(* IEC 61131-3 sources: elnaProjects/kc6/build_BaseProject_ecl/_ (part 2) *)

  StrAlg.CanRun := StrAlg.inCanRun;
  StrAlg.OpcCommandsDisabled := StrAlg.inOpcCommandsDisabled;

  IF StrAlg.isRuning THEN

      StrAlg.hasError := pnsOff.error OR nu1Off.error OR nu2Off.error
      OR stopNU1.error OR stopNU2.error OR testUnsuccessful.error;

      IF puskOilSystem.top THEN
           askQuestion(algContinue);
      END_IF;

      IF algContinue.answer = _Answers.ANS_YES AND NOT nuOff.top THEN

          runPhase(nuOff);

          IF Im.nu1.onStatus = _statusDualInput.STATUS_ON THEN
  		runPhase(nu1Off);
          END_IF;

          IF Im.nu2.onStatus = _statusDualInput.STATUS_ON THEN
  		runPhase(nu2Off);
          END_IF;

      END_IF;

      IF nuOff.start AND NOT nuOff.top THEN
            runPhase(BreakTest);
  	nuOff.top:= Im.nu1.onStatus = _statusDualInput.STATUS_Off
                    AND Im.nu2.onStatus = _statusDualInput.STATUS_Off;
      END_IF;

      IF nuOff.top THEN

          runPhase(dPmgAi);
          runPhase(dPmgDi);
      END_IF;

      IF dPmgDi.start AND NOT dPmgDi.top THEN
          dPmgDi.top:=Im.SingleSignals.dP_maslo_gaz_menshe_100_kPa.q;
      END_IF;

      IF dPmgAi.top AND dPmgDi.top THEN
          runPhase(nuOn);
          runPhase(noRezrv);
      END_IF;

      IF noRezrv.start AND NOT noRezrv.top THEN
          noRezrv.top:=NotHasRezervNU;
      END_IF;

       IF nuOn.start AND (NOT WaitOnNU.Q) THEN
          WaitOnNU(IN:=Im.nu1.onStatus = _statusDualInput.STATUS_On OR
              Im.nu2.onStatus = _statusDualInput.STATUS_On, PT:=T#1S);
          nuOn.top:=Im.nu1.onStatus = _statusDualInput.STATUS_On OR
              Im.nu2.onStatus = _statusDualInput.STATUS_On;
      END_IF;

      IF  WaitOnNU.Q AND noRezrv.top THEN
          ai.Perepad_davleniya_maslo_gaz.Disabled_LA:=TRUE;
          ai.Perepad_davleniya_maslo_gaz.Disabled_LW:=TRUE;
          ai.Davlenie_masla_smazki_nizkoe.Disabled_LA:=TRUE;
          ai.Davlenie_masla_smazki_nizkoe.Disabled_LW:=TRUE;
          ai.Davlenie_masla_smazki_visokoe.Disabled_LW:=TRUE;

          resetAiProtection(protections.Davlenie_masla_smazki_nizkoe_LA);
          resetAiProtection(protections.Perepad_davleniya_maslo_gaz_LA);
          resetDiProtection(protections.dP_maslo_gaz_menshe_100_kPa_DI);

          resetIfRunning(algoritms.autoNu);
          resetIfRunning(algoritms.AutoPns);

          runPhase(stopANU);
          runPhase(pnsOff);

          runPhase(stopNU1);
          runPhase(stopNU2);

      END_IF;

      IF stopANU.start AND NOT stopANU.top THEN

  	stopANU.top:= Im.nu1.onStatus = _statusDualInput.STATUS_Off AND
                          Im.nu2.onStatus = _statusDualInput.STATUS_Off;
      END_IF;

      IF BreakTest.top AND NOT pnsOff.top THEN
  	testUnsuccessful.error:=TRUE;
      END_IF;

      IF pnsOff.top AND stopANU.top THEN
            resetPhase(BreakTest);
  	waitReset(IN:=TRUE, PT:= T#3S);
      END_IF;

      IF waitReset.Q THEN
          algManager.nMode:=ModeGpa.MODE_STOP;
          resetIfRunning(StrAlg);
      END_IF;

      StrAlg.isEnded:= pnsOff.top AND stopANU.top;

  END_IF;

  StrAlg.CanRun := StrAlg.inCanRun;
  StrAlg.OpcCommandsDisabled := StrAlg.inOpcCommandsDisabled;

  (* ---- Если управление с ВУ заблокировано, то  передаем команду из алгоритма ---- *)
  IF StrAlg.inOpcCommandsDisabled THEN
  	StrAlg.inCommand := StrAlg.inCommand_Alg;
  ELSE (* иначе передаем команду с АРМа*)
  	StrAlg.inCommand := StrAlg.inCommand_ARM;
  END_IF;

  _sunpackerCommand(command := StrAlg.inCommand);
  	source := _sunpackerCommand.source;
  	cmd := _sunpackerCommand.cmd;

  IF cmd <> 0 AND lastCmd <> cmd AND (((NOT StrAlg.opcCommandsDisabled) AND source > 0) OR source = 0) then
  	CASE BYTE_TO_INT(cmd) OF
  		(*cmdRun*) 1: 	IF (StrAlg.CanRun) THEN
  					StrAlg.isRuning := TRUE;
  					StrAlg.isEnded := FALSE;
  					StrAlg.hasError := FALSE;
  					(*****************       OnRun       *****************)

                                                    algManager.nMode:=ModeGpa.MODE_TESTDPMG;
                                                    algoritms.puskOilSystem.inCanRun:= TRUE;
                                                    runPhase(puskOilSystem);

  					cmd_for_Status := cmd;
  					source_for_Status := source;
  					command_error_for_Status := 0;
  				ELSE
  					StrAlg.isRuning := FALSE;
  					StrAlg.isEnded := FALSE;
  					StrAlg.hasError 	:= FALSE;

  					cmd_for_Status := 0;
  					source_for_Status := source;
  					command_error_for_Status := cmd;
  				END_IF;
  		(*cmdReset*) 2: 	StrAlg.isRuning := FALSE;
  				StrAlg.isEnded := FALSE;
  				StrAlg.hasError 	:= FALSE;

                                           (*****************       OnReset       *****************)
                                          waitReset(IN:=FALSE);
                                          WaitOnNU(IN:=FALSE);

                                          ai.Davlenie_masla_smazki_nizkoe.Disabled_LA:=TRUE;
                                          ai.Davlenie_masla_smazki_nizkoe.Disabled_LW:=TRUE;
                                          ai.Davlenie_masla_smazki_visokoe.Disabled_LW:=TRUE;
                                          resetAiProtection(protections.Davlenie_masla_smazki_nizkoe_LA);
                                          resetAiProtection(protections.Perepad_davleniya_maslo_gaz_LA);
                                          resetDiProtection(protections.dP_maslo_gaz_menshe_100_kPa_DI);

                                          resetPhase(puskOilSystem);
                                          resetPhase(nuOff);
                                          resetPhase(dPmgAi);
                                          resetPhase(dPmgDi);
                                          resetPhase(nuOn);
                                          resetPhase(noRezrv);
                                          resetPhase(BreakTest);
                                          resetPhase(testUnsuccessful);
                                          resetPhase(pnsOff);
                                          resetPhase(stopANU);
                                          resetPhase(nu1Off);
                                          resetPhase(nu2Off);
                                          resetPhase(stopNU1);
                                          resetPhase(stopNU2);

                                          resetQuestion(algContinue);

  				cmd_for_Status := cmd;
  				source_for_Status := source;
  				command_error_for_Status := 0;
  	END_CASE;
  	resetCmdTimer(IN := false);
  	resetCmdTimerPriznak := TRUE;
  END_IF;
  lastCmd := cmd;

  resetCmdTimer(IN := resetCmdTimerPriznak, PT := T#5S);
  IF resetCmdTimer.Q THEN
  	resetCmdTimerPriznak := FALSE;
  	source_for_Status := 0;
  	cmd_for_Status := 0;
  	command_error_for_Status := 0;
  END_IF;

  StrAlg.Start:= puskOilSystem.startStatus
              OR nuOff.startStatus
              OR dPmgAi.startStatus
              OR dPmgDi.startStatus
              OR nuOn.startStatus
              OR noRezrv.startStatus
              OR BreakTest.startStatus
              OR testUnsuccessful.startStatus
              OR pnsOff.startStatus
              OR stopANU.startStatus
              OR nu1Off.startStatus
              OR nu2Off.startStatus;

  StrAlg.Error:=  puskOilSystem.errorStatus
              OR nuOff.errorStatus
              OR dPmgAi.errorStatus
              OR dPmgDi.errorStatus
              OR nuOn.errorStatus
              OR noRezrv.errorStatus
              OR BreakTest.errorStatus
              OR testUnsuccessful.errorStatus
              OR pnsOff.errorStatus
              OR stopANU.errorStatus
              OR nu1Off.errorStatus
              OR nu2Off.errorStatus;

  StrAlg.Top:=   puskOilSystem.topStatus
              OR nuOff.topStatus
              OR dPmgAi.topStatus
              OR dPmgDi.topStatus
              OR nuOn.topStatus
              OR noRezrv.topStatus
              OR BreakTest.topStatus
              OR testUnsuccessful.topStatus
              OR pnsOff.topStatus
              OR stopANU.topStatus
              OR nu1Off.topStatus
              OR nu2Off.topStatus;

  (*TODO: TYPE PROGRAM CODE HERE*)
  StrAlg.status :=  SHL(BYTE_TO_DWORD(source_for_Status), 29)
  			OR SHL(BYTE_TO_DWORD(cmd_for_Status), 26)
  			OR SHL(BYTE_TO_DWORD(command_error_for_Status), 23)
  			OR SHL(BOOL_TO_DWORD(StrAlg.OpcCommandsDisabled ), 21)
  			OR SHL(BOOL_TO_DWORD(StrAlg.hasError),4)
  			OR SHL(BOOL_TO_DWORD(StrAlg.CanRun),2)
  			OR SHL(BOOL_TO_DWORD(StrAlg.isEnded),1)
  			OR BOOL_TO_DWORD(StrAlg.isRuning);
END_FUNCTION_BLOCK

FUNCTION_BLOCK fb_ph_DIprotection
  VAR_IN_OUT
    StrDiP : struct_DiProtection;
  END_VAR
  VAR_INPUT
    act : TYPE_PhaseAlgoritmAction;
    PhaseNumber : UINT;
  END_VAR
  VAR_IN_OUT
    StrPh : struct_PhaseAlgoritm;
  END_VAR
  VAR
    CommandFault_Trig : R_TRIG;
    reset_Trig : R_TRIG;
    _statusDualInput : TYPE_statusDualInput;
  END_VAR

  IF StrPh.run AND NOT StrPh.start THEN
  	StrPh.start := TRUE;
  	StrPh.top := FALSE;
  	StrPh.error := FALSE;
            StrPh.run:=FALSE;

  	CASE act OF
  		(*PhaseAlgoritmAction.run*)    _run : runDiProtection(StrDiP); (*cmd_run*)
  		(*PhaseAlgoritmAction.reset*)_reset : resetDiProtection(StrDiP); (*cmd_reset*)
  	END_CASE;
  END_IF;

  IF StrPh.start AND NOT StrPh.top THEN
                      CommandFault_Trig(CLK := StrDiP.hasError);
                      IF CommandFault_Trig.Q THEN
  	          StrPh.error := TRUE;
                      END_IF;

  		CASE act OF
  		(*PhaseAlgoritmAction.run*)    _run:    StrPh.top:=StrDiP.isRunning;

  		(*PhaseAlgoritmAction.reset*) _reset:   StrPh.top := NOT StrDiP.isRunning;
  		END_CASE;

  END_IF;

  IF StrPh.top THEN
  StrPh.error := FALSE;
  END_IF;

  reset_Trig(CLK := StrPh.reset);
  IF reset_Trig.Q THEN
            StrPh.start := FALSE;
  	StrPh.error := FALSE;
  	StrPh.top := FALSE;
            StrPh.run:=FALSE;
            StrPh.reset:=FALSE;
  END_IF;

  StrPh.startStatus := SHL(BOOL_TO_DWORD(StrPh.start), PhaseNumber);
  StrPh.errorStatus := SHL(BOOL_TO_DWORD(StrPh.error), PhaseNumber);
  StrPh.topStatus := SHL(BOOL_TO_DWORD(StrPh.top), PhaseNumber);
END_FUNCTION_BLOCK

FUNCTION_BLOCK fb_ph_Kran
  VAR_IN_OUT
    im : struct_Kran;
    StrPh : struct_PhaseAlgoritm;
  END_VAR
  VAR_INPUT
    act : TYPE_DualStateImAction;
    PhaseNumber : UINT;
  END_VAR
  VAR
    CommandFault_Trig : R_TRIG;
    reset_Trig : R_TRIG;
    _statusDualInput : TYPE_statusDualInput;
  END_VAR

  IF StrPh.run AND NOT StrPh.start THEN
  	StrPh.start := TRUE;
  	StrPh.top := FALSE;
  	StrPh.error := FALSE;
            StrPh.run:=FALSE;

  	CASE act OF
  		(*DualStateImAction.on*)   _on: im.inCommand_Alg := 1; (*cmd_open*)
  		(*DualStateImAction.off*) _off: im.inCommand_Alg := 2; (*cmd_close*)
  	END_CASE;
  END_IF;

  IF StrPh.start AND NOT StrPh.top THEN
                      CommandFault_Trig(CLK := im.CommandFault);
                      IF CommandFault_Trig.Q THEN
  	          StrPh.error := TRUE;
                      END_IF;

  		CASE act OF
  		(*_DualStateImAction.on*)    _on: StrPh.top := im.onStatus = _statusDualInput.STATUS_ON;
  		(*_DualStateImAction.off*)  _off: StrPh.top := im.onStatus = _statusDualInput.STATUS_OFF;
  		END_CASE;

  END_IF;

  IF StrPh.top THEN
  StrPh.error := FALSE;
  END_IF;

  reset_Trig(CLK := StrPh.reset);
  IF reset_Trig.Q THEN
  	StrPh.start := FALSE;
  	StrPh.error := FALSE;
  	StrPh.top := FALSE;
            StrPh.run:=FALSE;
            StrPh.reset:=FALSE;
  END_IF;

  StrPh.startStatus := SHL(BOOL_TO_DWORD(StrPh.start), PhaseNumber);
  StrPh.errorStatus := SHL(BOOL_TO_DWORD(StrPh.error), PhaseNumber);
  StrPh.topStatus := SHL(BOOL_TO_DWORD(StrPh.top), PhaseNumber);
END_FUNCTION_BLOCK

FUNCTION_BLOCK fb_ph_SectionSwitch
  VAR_IN_OUT
    im : struct_SectionSwitch;
  END_VAR
  VAR_INPUT
    act : TYPE_DualStateImAction;
    PhaseNumber : UINT;
  END_VAR
  VAR_IN_OUT
    StrPh : struct_PhaseAlgoritm;
  END_VAR
  VAR
    CommandFault_Trig : R_TRIG;
    reset_Trig : R_TRIG;
    _statusDualInput : TYPE_statusDualInput;
  END_VAR

  IF StrPh.run AND NOT StrPh.start THEN
  	StrPh.start := TRUE;
  	StrPh.top := FALSE;
  	StrPh.error := FALSE;
            StrPh.run:=FALSE;

  	CASE act OF
  		(*DualStateImAction.on*)   _on : im.inCommand_Alg := 1; (*cmd_open*)
  		(*DualStateImAction.off*) _off : im.inCommand_Alg := 2; (*cmd_close*)
  	END_CASE;
  END_IF;

  IF StrPh.start AND NOT StrPh.top THEN
                      CommandFault_Trig(CLK := im.CommandFault);
                      IF CommandFault_Trig.Q THEN
  	          StrPh.error := TRUE;
                      END_IF;

  		CASE act OF
  		(*_DualStateImAction.on*)    _on: StrPh.top := im.onStatus = _statusDualInput.STATUS_ON;
  		(*_DualStateImAction.off*)  _off: StrPh.top := im.onStatus = _statusDualInput.STATUS_OFF;
  		END_CASE;

  END_IF;

  IF StrPh.top THEN
  StrPh.error := FALSE;
  END_IF;

  reset_Trig(CLK := StrPh.reset);
  IF reset_Trig.Q THEN
  	StrPh.start := FALSE;
  	StrPh.error := FALSE;
  	StrPh.top := FALSE;
            StrPh.run:=FALSE;
            StrPh.reset:=FALSE;
  END_IF;

  StrPh.startStatus := SHL(BOOL_TO_DWORD(StrPh.start), PhaseNumber);
  StrPh.errorStatus := SHL(BOOL_TO_DWORD(StrPh.error), PhaseNumber);
  StrPh.topStatus := SHL(BOOL_TO_DWORD(StrPh.top), PhaseNumber);
END_FUNCTION_BLOCK

FUNCTION_BLOCK puskKalg
  VAR_IN_OUT
    StrAlg : struct_Alg;
  END_VAR
  VAR
    puskOilSystem : struct_PhaseAlgoritm;
  END_VAR
  VAR_IN_OUT
    questionFilling : struct_Question;
  END_VAR
  VAR
    filling : struct_PhaseAlgoritm;
  END_VAR
  VAR_IN_OUT
    questionUnload : struct_Question;
  END_VAR
  VAR
    kran3bOpen : struct_PhaseAlgoritm;
    kran4Close : struct_PhaseAlgoritm;
    kran1Close : struct_PhaseAlgoritm;
    kran2Close : struct_PhaseAlgoritm;
    kran5open : struct_PhaseAlgoritm;
    wait720 : struct_PhaseAlgoritm;
    noGasInPipe : struct_PhaseAlgoritm;
    AutoNUoff : struct_PhaseAlgoritm;
    nu1Off : struct_PhaseAlgoritm;
    nu2Off : struct_PhaseAlgoritm;
    pnsWaitOff : struct_PhaseAlgoritm;
    testUnsuccessfulUnfill : struct_PhaseAlgoritm;
    fb_puskOilSystem : fb_ph_algoritm;
    fb_questionFilling : fb_Question;
    fb_filling : fb_ph_algoritm;
    fb_questionUnload : fb_Question;
    fb_kran3bOpen : fb_ph_Kran;
    fb_kran4Close : fb_ph_CustomPhase;
    fb_kran1Close : fb_ph_Kran;
    fb_kran2Close : fb_ph_Kran;
    fb_kran5open : fb_ph_Kran;
    fb_wait720 : fb_ph_Timer;
    fb_noGasInPipe : fb_ph_CustomPhase;
    fb_AutoNUoff : fb_ph_algoritm;
    fb_nu1Off : fb_ph_OilPump;
    fb_nu2Off : fb_ph_OilPump;
    fb_pnsWaitOff : fb_ph_algoritm;
    fb_testUnsuccessfulUnfill : fb_ph_CustomPhase;
    _sunpackerCommand : fb_sunpackerCommand;
    _DualStateImAction : TYPE_DualStateImAction;
    _Answers : TYPE_Answers;
    _statusDualInput : TYPE_statusDualInput;
    _StatusAi : TYPE_StatusAi;
    _PhaseAlgoritmAction : TYPE_PhaseAlgoritmAction;
    source : BYTE;
    cmd : BYTE;
    lastCmd : BYTE;
    source_for_Status : BYTE;
    cmd_for_Status : BYTE;
    command_error_for_Status : BYTE;
    resetCmdTimer : TON;
    resetCmdTimerPriznak : BOOL;
    testKranControl : BOOL      := TRUE;
    onInit : BOOL;
    waitReset : TON;
  END_VAR
  VAR_EXTERNAL
    IM : ImConfig;
    algoritms : AlgoritmsConfig;
    ai : AiConfig;
    AlgTimers : struct_AlgTimers;
    ModeGpa : TYPE_ModeGpa;
    algManager : struct_AlgoritmsManager;
    protections : ProtectionsConfig;
  END_VAR
  VAR CONSTANT
    Ust_Pgaza : LREAL      := 0.3;
  END_VAR

  IF NOT onInit THEN

            fb_puskOilSystem(phaseNumber:=0, act:=_run, waitCompletion:=TRUE);
        questionFilling.AnswerVariants:=_Answers.ANS_YES;
                  fb_filling(phaseNumber:=1, act:=_run, waitCompletion:=TRUE);
      questionUnload.AnswerVariants:=_Answers.ANS_YES;
               fb_kran3bOpen(phaseNumber:=3, act:=_on);
               fb_kran4Close(phaseNumber:=4);
               fb_kran1Close(phaseNumber:=5, act:=_off);
               fb_kran2Close(phaseNumber:=6, act:=_off);
                fb_kran5open(phaseNumber:=7, act:=_on);
                  fb_wait720(phaseNumber:=8, delay:=T#720S);
              fb_noGasInPipe(phaseNumber:=9);
                fb_AutoNUoff(phaseNumber:=10, act:=_reset, waitCompletion:=FALSE);
                   fb_nu1Off(phaseNumber:=11, act:=_off);
                   fb_nu2Off(phaseNumber:=12, act:=_off);
               fb_pnsWaitOff(phaseNumber:=15, act:=_run, waitCompletion:=TRUE);
   fb_testUnsuccessfulUnfill(phaseNumber:=18);

  onInit:=TRUE;
  END_IF;

            fb_puskOilSystem(StrPh:=puskOilSystem, alg:=algoritms.puskOilSystem);
          fb_questionFilling(StrQ:=questionFilling);
                  fb_filling(StrPh:=filling, alg:=algoritms.filling);
           fb_questionUnload(StrQ:=questionUnload);
               fb_kran3bOpen(StrPh:=kran3bOpen, Im:=Im.kran3b);
               fb_kran4Close(StrPh:=kran4Close);
               fb_kran1Close(StrPh:=kran1Close, Im:=Im.kran1);
               fb_kran2Close(StrPh:=kran2Close, Im:=Im.kran2);
                fb_kran5open(StrPh:=kran5open, Im:=Im.kran5);
                  fb_wait720(StrPh:=wait720, timer:=AlgTimers.puskK_wait720);
              fb_noGasInPipe(StrPh:=noGasInPipe);
                fb_AutoNUoff(StrPh:=AutoNUoff, alg:=algoritms.autoNu);
                   fb_nu1Off(StrPh:=nu1Off, Im:=Im.nu1);
                   fb_nu2Off(StrPh:=nu2Off, Im:=Im.nu2);
               fb_pnsWaitOff(StrPh:=pnsWaitOff, alg:=algoritms.vibegPNS);
   fb_testUnsuccessfulUnfill(StrPh:=testUnsuccessfulUnfill);

  StrAlg.CanRun := StrAlg.inCanRun;
  StrAlg.OpcCommandsDisabled := StrAlg.inOpcCommandsDisabled;

  IF StrAlg.isRuning THEN

      StrAlg.hasError := kran3bOpen.error OR kran1Close.error OR kran2Close.error OR kran5open.error OR testUnsuccessfulUnfill.error;

      IF puskOilSystem.top THEN
           askQuestion(questionFilling);
      END_IF;

      IF questionFilling.answer = _Answers.ANS_YES THEN
          runPhase(filling);
      END_IF;

      IF filling.top THEN
         askQuestion(questionUnload);
      END_IF;

       IF questionUnload.answer = _Answers.ANS_YES THEN
          runPhase(kran3bOpen);
          runPhase(wait720);
      END_IF;

      IF kran3bOpen.top THEN
            resetDiProtection(protections.Kran1sdvig);
            resetDiProtection(protections.Kran2sdvig);

            runPhase(kran1Close);
            runPhase(kran2Close);
            runPhase(kran4Close);
      END_IF;

       IF kran4Close.start AND NOT kran4Close.top THEN
  	kran4Close.top:= Im.kran4.onStatus = _statusDualInput.STATUS_OFF;
      END_IF;

      IF kran1Close.top AND kran2Close.top AND kran4Close.top THEN
  	runPhase(kran5open);
      END_IF;

      IF kran5open.top THEN
  	runPhase(noGasInPipe);
      END_IF;

      IF noGasInPipe.start AND (NOT noGasInPipe.top) THEN
  	noGasInPipe.top:=  (ai.Davlenie_gaza_na_vhode_nagnetatelya.interval >= _statusAi.NORMAL
                           AND  ai.Davlenie_gaza_na_vhode_nagnetatelya.value< Ust_Pgaza )
                           AND (ai.Davlenie_gaza_na_vihode_nagnetatelya.interval >= _statusAi.NORMAL
                           AND  ai.Davlenie_gaza_na_vihode_nagnetatelya.value< Ust_Pgaza);
      END_IF;

      IF noGasInPipe.top THEN

            ai.Perepad_davleniya_maslo_gaz.Disabled_LA:=TRUE;
            ai.Perepad_davleniya_maslo_gaz.Disabled_LW:=TRUE;
            resetAiProtection(protections.Perepad_davleniya_maslo_gaz_LA);
            resetDiProtection(protections.dP_maslo_gaz_menshe_100_kPa_DI);
  	runPhase(AutoNUoff);

      END_IF;

       IF autoNuOff.top THEN
  	runPhase(nu1off);
            runPhase(nu2off);
      END_IF;

      IF nu1Off.top AND nu2Off.top THEN
  	runPhase(pnsWaitOff);
      END_IF;

      IF wait720.top AND NOT (pnsWaitOff.top) THEN
            testUnsuccessfulUnfill.error:=TRUE;
      END_IF;

      IF pnsWaitOff.top THEN
            resetPhase(wait720);
  	waitReset(IN:=TRUE, PT:= T#2S);
      END_IF;

      IF waitReset.Q THEN
          resetIfRunning(algoritms.vibegPNS);
          algManager.nMode:=ModeGpa.MODE_STOP;
          resetIfRunning(StrAlg);
      END_IF;

      StrAlg.isEnded:= nu1Off.top AND nu2Off.top;

      IF testKranControl THEN
  	IF      (im.pns.onStatus = _statusDualInput.STATUS_ON)
                AND (im.nu1.onStatus = _statusDualInput.STATUS_ON OR im.nu2.onStatus = _statusDualInput.STATUS_ON)
  	    AND (ai.Perepad_davleniya_maslo_gaz.interval >= _statusAi.normal)
                AND (ai.Perepad_davleniya_maslo_gaz.value > im.PuskOilSystem_UstdPmg.Value)
            THEN
  	    IM.Kran3b.inOpcCommandsDisabled:=FALSE;
  	    Im.kran4.inOpcCommandsDisabled:=FALSE;
  	    Im.kran5.inOpcCommandsDisabled:=FALSE;
  		IF	Im.SingleSignals.dP_gaza_kr_1.q THEN
  			Im.kran1.inOpcCommandsDisabled:=FALSE;
  			Im.kran2.inOpcCommandsDisabled:=FALSE;
  		ELSE
  			Im.kran1.inOpcCommandsDisabled:=TRUE;
  			Im.kran2.inOpcCommandsDisabled:=TRUE;
  		END_IF;
            ELSE
  	    Im.kran1.inOpcCommandsDisabled:=TRUE;
  	    Im.kran2.inOpcCommandsDisabled:=TRUE;
  	    Im.kran3b.inOpcCommandsDisabled:=TRUE;
  	    Im.kran4.inOpcCommandsDisabled:=TRUE;
  	    Im.kran5.inOpcCommandsDisabled:=TRUE;
            END_IF;

      ELSE
  	Im.kran1.inOpcCommandsDisabled:=TRUE;
  	Im.kran2.inOpcCommandsDisabled:=TRUE;
  	Im.kran3b.inOpcCommandsDisabled:=TRUE;
  	Im.kran4.inOpcCommandsDisabled:=TRUE;
  	Im.kran5.inOpcCommandsDisabled:=TRUE;
      END_IF;
  END_IF;

  StrAlg.CanRun := StrAlg.inCanRun;
  StrAlg.OpcCommandsDisabled := StrAlg.inOpcCommandsDisabled;

  (* ---- Если управление с ВУ заблокировано, то  передаем команду из алгоритма ---- *)
  IF StrAlg.inOpcCommandsDisabled THEN
  	StrAlg.inCommand := StrAlg.inCommand_Alg;
  ELSE (* иначе передаем команду с АРМа*)
  	StrAlg.inCommand := StrAlg.inCommand_ARM;
  END_IF;

  _sunpackerCommand(command := StrAlg.inCommand);
  	source := _sunpackerCommand.source;
  	cmd := _sunpackerCommand.cmd;

  IF cmd <> 0 AND lastCmd <> cmd AND (((NOT StrAlg.opcCommandsDisabled) AND source > 0) OR source = 0) then
  	CASE BYTE_TO_INT(cmd) OF
  		(*cmdRun*) 1: 	IF (StrAlg.CanRun) THEN
  					StrAlg.isRuning := TRUE;
  					StrAlg.isEnded := FALSE;
  					StrAlg.hasError := FALSE;
  					(*****************       OnRun       *****************)

                                                    algManager.nMode:=ModeGpa.MODE_PUSKK;
                                                    algoritms.puskOilSystem.inCanRun:= TRUE;
                                                    algoritms.filling.inCanRun:= TRUE;
                                                    runPhase(puskOilSystem);

  					cmd_for_Status := cmd;
  					source_for_Status := source;
  					command_error_for_Status := 0;
  				ELSE
  					StrAlg.isRuning := FALSE;
  					StrAlg.isEnded := FALSE;
  					StrAlg.hasError 	:= FALSE;

  					cmd_for_Status := 0;
  					source_for_Status := source;
  					command_error_for_Status := cmd;
  				END_IF;
  		(*cmdReset*) 2: 	StrAlg.isRuning := FALSE;
  				StrAlg.isEnded := FALSE;
  				StrAlg.hasError 	:= FALSE;

                                           (*****************       OnReset       *****************)
                                          (*testKranControl:=FALSE;*)
                                          waitReset(IN:=FALSE);

                                          resetPhase(puskOilSystem);
                                          resetPhase(filling);
                                          resetPhase(kran3bOpen);
                                          resetPhase(kran4Close);
                                          resetPhase(kran1Close);
                                          resetPhase(kran2Close);
                                          resetPhase(kran5open);
                                          resetPhase(wait720);
                                          resetPhase(noGasInPipe);
                                          resetPhase(AutoNUoff);
                                          resetPhase(nu1Off);
                                          resetPhase(nu2Off);
                                          resetPhase(pnsWaitOff);
                                          resetPhase(testUnsuccessfulUnfill);
                                          BlockAllIM(IM);
                                          resetQuestion(questionFilling);
                                          resetQuestion(questionUnload);

  				cmd_for_Status := cmd;
  				source_for_Status := source;
  				command_error_for_Status := 0;
  	END_CASE;
  	resetCmdTimer(IN := false);
  	resetCmdTimerPriznak := TRUE;
  END_IF;
  lastCmd := cmd;

  resetCmdTimer(IN := resetCmdTimerPriznak, PT := T#5S);
  IF resetCmdTimer.Q THEN
  	resetCmdTimerPriznak := FALSE;
  	source_for_Status := 0;
  	cmd_for_Status := 0;
  	command_error_for_Status := 0;
  END_IF;

  StrAlg.Start:= puskOilSystem.startStatus
              OR filling.startStatus
              OR kran3bOpen.startStatus
              OR kran4Close.startStatus
              OR kran1Close.startStatus
              OR kran2Close.startStatus
              OR kran5open.startStatus
              OR wait720.startStatus
              OR noGasInPipe.startStatus
              OR AutoNUoff.startStatus
              OR nu1Off.startStatus
              OR nu2Off.startStatus
              OR pnsWaitOff.startStatus
              OR testUnsuccessfulUnfill.startStatus;

  StrAlg.Error:=  puskOilSystem.errorStatus
              OR filling.errorStatus
              OR kran3bOpen.errorStatus
              OR kran4Close.errorStatus
              OR kran1Close.errorStatus
              OR kran2Close.errorStatus
              OR kran5open.errorStatus
              OR wait720.errorStatus
              OR noGasInPipe.errorStatus
              OR AutoNUoff.errorStatus
              OR nu1Off.errorStatus
              OR nu2Off.errorStatus
              OR pnsWaitOff.errorStatus
              OR testUnsuccessfulUnfill.errorStatus;

  StrAlg.Top:=   puskOilSystem.topStatus
              OR filling.topStatus
              OR kran3bOpen.topStatus
              OR kran4Close.topStatus
              OR kran1Close.topStatus
              OR kran2Close.topStatus
              OR kran5open.topStatus
              OR wait720.topStatus
              OR noGasInPipe.topStatus
              OR AutoNUoff.topStatus
              OR nu1Off.topStatus
              OR nu2Off.topStatus
              OR pnsWaitOff.topStatus
              OR testUnsuccessfulUnfill.topStatus;

  (*TODO: TYPE PROGRAM CODE HERE*)
  StrAlg.status :=  SHL(BYTE_TO_DWORD(source_for_Status), 29)
  			OR SHL(BYTE_TO_DWORD(cmd_for_Status), 26)
  			OR SHL(BYTE_TO_DWORD(command_error_for_Status), 23)
  			OR SHL(BOOL_TO_DWORD(StrAlg.OpcCommandsDisabled ), 21)
  			OR SHL(BOOL_TO_DWORD(StrAlg.hasError),4)
  			OR SHL(BOOL_TO_DWORD(StrAlg.CanRun),2)
  			OR SHL(BOOL_TO_DWORD(StrAlg.isEnded),1)
  			OR BOOL_TO_DWORD(StrAlg.isRuning);
END_FUNCTION_BLOCK

FUNCTION_BLOCK puskValg
  VAR_IN_OUT
    StrAlg : struct_Alg;
  END_VAR
  VAR
    puskOilSystem : struct_PhaseAlgoritm;
  END_VAR
  VAR_IN_OUT
    questionEngine : struct_Question;
  END_VAR
  VAR
    runningEngine : struct_PhaseAlgoritm;
  END_VAR
  VAR_IN_OUT
    questionMVoff : struct_Question;
  END_VAR
  VAR
    mvOff : struct_PhaseAlgoritm;
    pnsOn : struct_PhaseAlgoritm;
    wait600 : struct_PhaseAlgoritm;
    AutoNUoff : struct_PhaseAlgoritm;
    nu1Off : struct_PhaseAlgoritm;
    nu2Off : struct_PhaseAlgoritm;
    Avom1Off : struct_PhaseAlgoritm;
    Avom2Off : struct_PhaseAlgoritm;
    pnsWaitOff : struct_PhaseAlgoritm;
    testUnsuccessful : struct_PhaseAlgoritm;
    fb_puskOilSystem : fb_ph_algoritm;
    fb_questionEngine : fb_Question;
    fb_runningEngine : fb_ph_algoritm;
    fb_questionMVoff : fb_Question;
    fb_mvOff : fb_ph_SectionSwitch;
    fb_pnsOn : fb_ph_Switch;
    fb_wait600 : fb_ph_Timer;
    fb_AutoNUoff : fb_ph_algoritm;
    fb_nu1Off : fb_ph_OilPump;
    fb_nu2Off : fb_ph_OilPump;
    fb_Avom1Off : fb_ph_Switch;
    fb_Avom2Off : fb_ph_Switch;
    fb_pnsWaitOff : fb_ph_algoritm;
    fb_testUnsuccessful : fb_ph_CustomPhase;
    _sunpackerCommand : fb_sunpackerCommand;
    _DualStateImAction : TYPE_DualStateImAction;
    _Answers : TYPE_Answers;
    _statusDualInput : TYPE_statusDualInput;
    _StatusAi : TYPE_StatusAi;
    _PhaseAlgoritmAction : TYPE_PhaseAlgoritmAction;
    source : BYTE;
    cmd : BYTE;
    lastCmd : BYTE;
    source_for_Status : BYTE;
    cmd_for_Status : BYTE;
    command_error_for_Status : BYTE;
    resetCmdTimer : TON;
    resetCmdTimerPriznak : BOOL;
    onInit : BOOL;
    waitReset : TON;
  END_VAR
  VAR_EXTERNAL
    IM : ImConfig;
    algoritms : AlgoritmsConfig;
    ai : AiConfig;
    AlgTimers : struct_AlgTimers;
    ModeGpa : TYPE_ModeGpa;
    algManager : struct_AlgoritmsManager;
    protections : ProtectionsConfig;
  END_VAR
  VAR CONSTANT
    Ust_Pgaza : LREAL      := 0.3;
  END_VAR

  IF NOT onInit THEN

            fb_puskOilSystem(phaseNumber:=0, act:=_run, waitCompletion:=TRUE);
         questionEngine.AnswerVariants:=_Answers.ANS_YES;
            fb_runningEngine(phaseNumber:=1, act:=_run, waitCompletion:=TRUE);
          questionMVoff.AnswerVariants:=_Answers.ANS_YES;
                    fb_mvOff(phaseNumber:=3, act:=_off);
                    fb_pnsOn(phaseNumber:=4, act:=_on);
                  fb_wait600(phaseNumber:=8, delay:=T#600S);
                fb_AutoNUoff(phaseNumber:=10, act:=_reset, waitCompletion:=FALSE);
                   fb_nu1Off(phaseNumber:=11, act:=_off);
                   fb_nu2Off(phaseNumber:=12, act:=_off);
               fb_pnsWaitOff(phaseNumber:=15, act:=_run, waitCompletion:=TRUE);
                 fb_Avom1Off(phaseNumber:=5, act:=_off);
                 fb_Avom2Off(phaseNumber:=6, act:=_off);
         fb_testUnsuccessful(phaseNumber:=17);

  onInit:=TRUE;
  END_IF;

            fb_puskOilSystem(StrPh:=puskOilSystem, alg:=algoritms.puskOilSystem);
           fb_questionEngine(StrQ:=questionEngine);
            fb_runningEngine(StrPh:=runningEngine, alg:=algoritms.filling);
            fb_questionMVoff(StrQ:=questionMVoff);
                    fb_mvOff(StrPh:=mvOff, Im:=Im.MB);
                    fb_pnsOn(StrPh:=pnsOn, Im:=Im.pns);
                  fb_wait600(StrPh:=wait600, timer:=AlgTimers.puskV_wait600);
                fb_AutoNUoff(StrPh:=AutoNUoff, alg:=algoritms.autoNu);
                   fb_nu1Off(StrPh:=nu1Off, Im:=Im.nu1);
                   fb_nu2Off(StrPh:=nu2Off, Im:=Im.nu2);
               fb_pnsWaitOff(StrPh:=pnsWaitOff, alg:=algoritms.vibegPNS);
                 fb_Avom1Off(StrPh:=Avom1Off, Im:=Im.v1_Avom);
                 fb_Avom2Off(StrPh:=Avom2Off, Im:=Im.v2_Avom);
         fb_testUnsuccessful(StrPh:=testUnsuccessful);

  StrAlg.CanRun := StrAlg.inCanRun;
  StrAlg.OpcCommandsDisabled := StrAlg.inOpcCommandsDisabled;

  IF StrAlg.isRuning THEN

      StrAlg.hasError := mvOff.error OR pnsOn.error OR testUnsuccessful.error;

      IF puskOilSystem.top THEN
           askQuestion(questionEngine);
      END_IF;

      IF questionEngine.answer = _Answers.ANS_YES THEN
          runPhase(runningEngine);
      END_IF;

      IF runningEngine.top THEN
         askQuestion(questionMVoff);
      END_IF;

       IF questionMVoff.answer = _Answers.ANS_YES THEN

          resetDiProtection(protections.MB);
          resetIfRunning(algoritms.AutoPns);
          runPhase(mvOff);
          runPhase(wait600);

       END_IF;

      IF mvOff.top THEN
          runPhase(pnsOn);
      END_IF;

      IF pnsOn.top THEN

            ai.Perepad_davleniya_maslo_gaz.Disabled_LA:=TRUE;
            ai.Perepad_davleniya_maslo_gaz.Disabled_LW:=TRUE;
            resetAiProtection(protections.Perepad_davleniya_maslo_gaz_LA);
            resetDiProtection(protections.dP_maslo_gaz_menshe_100_kPa_DI);
  	runPhase(AutoNUoff);

      END_IF;

       IF autoNuOff.top THEN
  	runPhase(nu1off);
            runPhase(nu2off);
      END_IF;

      IF nu1Off.top AND nu2Off.top THEN
  	runPhase(pnsWaitOff);
      END_IF;

      IF wait600.top AND NOT (pnsWaitOff.top) THEN
            testUnsuccessful.error:=TRUE;
      END_IF;

      IF pnsWaitOff.top THEN
            resetPhase(wait600);
            resetIfRunning(algoritms.AutoAvom);
            runPhase(Avom1Off);
            runPhase(Avom2Off);
  	waitReset(IN:=TRUE, PT:= T#2S);
      END_IF;

      IF waitReset.Q THEN
          resetIfRunning(algoritms.vibegPNS);
          algManager.nMode:=ModeGpa.MODE_STOP;
          resetIfRunning(StrAlg);
      END_IF;

      StrAlg.isEnded:= pnsWaitOff.top;

  END_IF;

  StrAlg.CanRun := StrAlg.inCanRun;
  StrAlg.OpcCommandsDisabled := StrAlg.inOpcCommandsDisabled;

  (* ---- Если управление с ВУ заблокировано, то  передаем команду из алгоритма ---- *)
  IF StrAlg.inOpcCommandsDisabled THEN
  	StrAlg.inCommand := StrAlg.inCommand_Alg;
  ELSE (* иначе передаем команду с АРМа*)
  	StrAlg.inCommand := StrAlg.inCommand_ARM;
  END_IF;

  _sunpackerCommand(command := StrAlg.inCommand);
  	source := _sunpackerCommand.source;
  	cmd := _sunpackerCommand.cmd;

  IF cmd <> 0 AND lastCmd <> cmd AND (((NOT StrAlg.opcCommandsDisabled) AND source > 0) OR source = 0) then
  	CASE BYTE_TO_INT(cmd) OF
  		(*cmdRun*) 1: 	IF (StrAlg.CanRun) THEN
  					StrAlg.isRuning := TRUE;
  					StrAlg.isEnded := FALSE;
  					StrAlg.hasError := FALSE;
  					(*****************       OnRun       *****************)

                                                    algManager.nMode:=ModeGpa.MODE_PUSKV;
                                                    algoritms.puskOilSystem.inCanRun:= TRUE;
                                                    algoritms.engineRun.inCanRun:= TRUE;
                                                    runPhase(puskOilSystem);

  					cmd_for_Status := cmd;
  					source_for_Status := source;
  					command_error_for_Status := 0;
  				ELSE
  					StrAlg.isRuning := FALSE;
  					StrAlg.isEnded := FALSE;
  					StrAlg.hasError 	:= FALSE;

  					cmd_for_Status := 0;
  					source_for_Status := source;
  					command_error_for_Status := cmd;
  				END_IF;
  		(*cmdReset*) 2: 	StrAlg.isRuning := FALSE;
  				StrAlg.isEnded := FALSE;
  				StrAlg.hasError 	:= FALSE;

                                           (*****************       OnReset       *****************)
                                          waitReset(IN:=FALSE);

                                          resetPhase(puskOilSystem);
                                          resetPhase(runningEngine);
                                          resetPhase(mvOff);
                                          resetPhase(pnsOn);
                                          resetPhase(wait600);
                                          resetPhase(AutoNUoff);
                                          resetPhase(nu1Off);
                                          resetPhase(nu2Off);
                                          resetPhase(pnsWaitOff);
                                          resetPhase(Avom1Off);
                                          resetPhase(Avom2Off);
                                          resetPhase(testUnsuccessful);

                                          resetQuestion(questionEngine);
                                          resetQuestion(questionMVoff);

  				cmd_for_Status := cmd;
  				source_for_Status := source;
  				command_error_for_Status := 0;
  	END_CASE;
  	resetCmdTimer(IN := false);
  	resetCmdTimerPriznak := TRUE;
  END_IF;
  lastCmd := cmd;

  resetCmdTimer(IN := resetCmdTimerPriznak, PT := T#5S);
  IF resetCmdTimer.Q THEN
  	resetCmdTimerPriznak := FALSE;
  	source_for_Status := 0;
  	cmd_for_Status := 0;
  	command_error_for_Status := 0;
  END_IF;

  StrAlg.Start:= puskOilSystem.startStatus
              OR runningEngine.startStatus
              OR mvOff.startStatus
              OR pnsOn.startStatus
              OR wait600.startStatus
              OR AutoNUoff.startStatus
              OR nu1Off.startStatus
              OR nu2Off.startStatus
              OR pnsWaitOff.startStatus
              OR testUnsuccessful.startStatus;

  StrAlg.Error:=  puskOilSystem.errorStatus
              OR runningEngine.errorStatus
              OR mvOff.errorStatus
              OR pnsOn.errorStatus
              OR wait600.errorStatus
              OR AutoNUoff.errorStatus
              OR nu1Off.errorStatus
              OR nu2Off.errorStatus
              OR pnsWaitOff.errorStatus
              OR testUnsuccessful.errorStatus;

  StrAlg.Top:=   puskOilSystem.topStatus
              OR runningEngine.topStatus
              OR mvOff.topStatus
              OR pnsOn.topStatus
              OR wait600.topStatus
              OR AutoNUoff.topStatus
              OR nu1Off.topStatus
              OR nu2Off.topStatus
              OR pnsWaitOff.topStatus
              OR testUnsuccessful.topStatus;

  (*TODO: TYPE PROGRAM CODE HERE*)
  StrAlg.status :=  SHL(BYTE_TO_DWORD(source_for_Status), 29)
  			OR SHL(BYTE_TO_DWORD(cmd_for_Status), 26)
  			OR SHL(BYTE_TO_DWORD(command_error_for_Status), 23)
  			OR SHL(BOOL_TO_DWORD(StrAlg.OpcCommandsDisabled ), 21)
  			OR SHL(BOOL_TO_DWORD(StrAlg.hasError),4)
  			OR SHL(BOOL_TO_DWORD(StrAlg.CanRun),2)
  			OR SHL(BOOL_TO_DWORD(StrAlg.isEnded),1)
  			OR BOOL_TO_DWORD(StrAlg.isRuning);
END_FUNCTION_BLOCK

FUNCTION_BLOCK AOAlg
  VAR_IN_OUT
    StrAlg : struct_Alg;
  END_VAR
  VAR
    kran4Close : struct_PhaseAlgoritm;
    mvOff : struct_PhaseAlgoritm;
    pnsOn : struct_PhaseAlgoritm;
    kran3bOpen : struct_PhaseAlgoritm;
    kran1Close : struct_PhaseAlgoritm;
    kran2Close : struct_PhaseAlgoritm;
    kran5Open : struct_PhaseAlgoritm;
    autoNuOff : struct_PhaseAlgoritm;
    autoPnsOff : struct_PhaseAlgoritm;
    pInNagLess100 : struct_PhaseAlgoritm;
    autoAvomOff : struct_PhaseAlgoritm;
    avom1cmdOff : struct_PhaseAlgoritm;
    avom2cmdOff : struct_PhaseAlgoritm;
    nu1off : struct_PhaseAlgoritm;
    nu2off : struct_PhaseAlgoritm;
    LowOil : struct_PhaseAlgoritm;
    waitKran : struct_PhaseAlgoritm;
    pnsWaitOff : struct_PhaseAlgoritm;
    runUnsuccessful : struct_PhaseAlgoritm;
    fb_kran4Close : fb_ph_Kran;
    fb_mvOff : fb_ph_SectionSwitch;
    fb_pnsOn : fb_ph_Switch;
    fb_kran3bOpen : fb_ph_Kran;
    fb_kran1Close : fb_ph_Kran;
    fb_kran2Close : fb_ph_Kran;
    fb_kran5Open : fb_ph_Kran;
    fb_autoNuOff : fb_ph_algoritm;
    fb_autoPnsOff : fb_ph_algoritm;
    fb_pInNagLess100 : fb_ph_CustomPhase;
    fb_autoAvomOff : fb_ph_algoritm;
    fb_avom1cmdOff : fb_ph_Switch;
    fb_avom2cmdOff : fb_ph_Switch;
    fb_nu1off : fb_ph_OilPump;
    fb_nu2off : fb_ph_OilPump;
    fb_LowOil : fb_ph_WaitAnalogValue;
    fb_waitKran : fb_ph_Timer;
    fb_pnsWaitOff : fb_ph_algoritm;
    fb_runUnsuccessful : fb_ph_CustomPhase;
    _sunpackerCommand : fb_sunpackerCommand;
    _statusAi : TYPE_StatusAi;
    _Answers : TYPE_Answers;
    _statusDualInput : TYPE_statusDualInput;
    _commandDualInput : TYPE_commandDualInput;
    _DualStateImAction : TYPE_DualStateImAction;
    _PhaseAlgoritmAction : TYPE_PhaseAlgoritmAction;
    source : BYTE;
    cmd : BYTE;
    lastCmd : BYTE;
    source_for_Status : BYTE;
    cmd_for_Status : BYTE;
    command_error_for_Status : BYTE;
    resetCmdTimer : TON;
    resetCmdTimerPriznak : BOOL;
    onInit : BOOL;
    waitReset : TON;
  END_VAR
  VAR_EXTERNAL
    IM : ImConfig;
    algoritms : AlgoritmsConfig;
    ai : AiConfig;
    protections : ProtectionsConfig;
    ModeGpa : TYPE_ModeGpa;
    algManager : struct_AlgoritmsManager;
    AlgTimers : struct_AlgTimers;
    PMcommand : TYPE_CommandsPotectionsManager;
    protectManager : struct_ProtectionsManager;
  END_VAR
  VAR CONSTANT
    Ust_Pgaza : LREAL      := 0.3;
  END_VAR

  IF NOT onInit THEN

         fb_kran4Close(phaseNumber:=1, act:=_off);
         fb_kran3bOpen(phaseNumber:=2, act:=_on);
              fb_mvOff(phaseNumber:=3, act:=_off);
              fb_pnsOn(phaseNumber:=4, act:=_on);
         fb_kran1Close(phaseNumber:=6, act:=_off);
         fb_kran2Close(phaseNumber:=7, act:=_off);
          fb_kran5Open(phaseNumber:=8, act:=_on);
          fb_autoNuOff(phaseNumber:=9, act:=_reset, waitCompletion:=FALSE);
         fb_autoPnsOff(phaseNumber:=10, act:=_reset, waitCompletion:=FALSE);
        fb_autoAvomOff(phaseNumber:=11, act:=_reset, waitCompletion:=FALSE);
        fb_avom1cmdOff(phaseNumber:=12, act:=_off);
        fb_avom2cmdOff(phaseNumber:=13, act:=_off);
      fb_pInNagLess100(phaseNumber:=14);
           fb_waitKran(phaseNumber:=15, delay:=T#240S);
         fb_pnsWaitOff(phaseNumber:=17, act:=_run, waitCompletion:=TRUE);
             fb_nu1off(phaseNumber:=18, act:=_off);
             fb_nu2off(phaseNumber:=19, act:=_off);
    fb_runUnsuccessful(phaseNumber:=20);

  onInit:=TRUE;
  END_IF;

         fb_kran4Close(StrPh:=kran4Close, Im:=Im.kran4);
         fb_kran3bOpen(StrPh:=kran3bOpen, Im:=Im.kran3b);
              fb_mvOff(StrPh:=mvOff, Im:=Im.MB);
              fb_pnsOn(StrPh:=pnsOn, Im:=Im.pns);

         fb_kran1Close(StrPh:=kran1Close, Im:=Im.kran1);
         fb_kran2Close(StrPh:=kran2Close, Im:=Im.kran2);
          fb_kran5Open(StrPh:=kran5Open, Im:=Im.kran5);
          fb_autoNuOff(StrPh:=autoNuOff, alg:=algoritms.autoNu);
         fb_autoPnsOff(StrPh:=autoPnsOff, alg:=algoritms.autoPns);
        fb_autoAvomOff(StrPh:=autoAvomOff, alg:=algoritms.AutoAvom);
        fb_avom1cmdOff(StrPh:=avom1cmdOff, Im:=Im.v1_Avom);
        fb_avom2cmdOff(StrPh:=avom2cmdOff, Im:=Im.v2_Avom);
      fb_pInNagLess100(StrPh:=pInNagLess100);
           fb_waitKran(StrPh:=waitKran, timer:=AlgTimers.AO_waitKran);
         fb_pnsWaitOff(StrPh:=pnsWaitOff, alg:=algoritms.vibegPNS, waitCompletion:=TRUE);
             fb_nu1off(StrPh:=nu1off, Im:=Im.nu1);
             fb_nu2off(StrPh:=nu2off, Im:=Im.nu2);
    fb_runUnsuccessful(StrPh:=runUnsuccessful);

  StrAlg.CanRun := StrAlg.inCanRun;
  StrAlg.OpcCommandsDisabled := StrAlg.inOpcCommandsDisabled;

  IF StrAlg.isRuning THEN

      StrAlg.hasError := kran4Close.error OR mvOff.error OR pnsOn.error OR kran3bOpen.error
      OR kran1Close.error OR kran2Close.error OR kran5Open.error OR runUnsuccessful.error;

      runPhase(kran4Close);
      runPhase(kran3bOpen);
      runPhase(kran1Close);
      runPhase(kran2Close);
      runPhase(mvOff);

      IF kran1Close.top AND kran2Close.top AND kran4Close.top THEN
          runPhase(kran5Open);
      END_IF;

      IF mvOff.top THEN
            runPhase(autoPnsOff);
      END_IF;

       IF autoPnsOff.top THEN
  	runPhase(pnsOn);
      END_IF;

      IF kran5Open.top THEN
         runPhase(pInNagLess100);
         resetPhase(waitKran);
      END_IF;

     IF pInNagLess100.start AND NOT pInNagLess100.top THEN
  	pInNagLess100.top:=( ai.Davlenie_gaza_na_vhode_nagnetatelya.interval >= _statusAi.NORMAL AND
            ai.Davlenie_gaza_na_vhode_nagnetatelya.value < Ust_Pgaza ) AND
           (ai.Davlenie_gaza_na_vihode_nagnetatelya.interval >= _statusAi.NORMAL AND
            ai.Davlenie_gaza_na_vihode_nagnetatelya.value < Ust_Pgaza);

     END_IF;

      IF pInNagLess100.top AND kran3bOpen.top AND mvOff.top THEN
  	ai.Perepad_davleniya_maslo_gaz.Disabled_LA:=TRUE;
            ai.Perepad_davleniya_maslo_gaz.Disabled_LW:=TRUE;
            resetAiProtection(protections.Perepad_davleniya_maslo_gaz_LA);
            resetDiProtection(protections.dP_maslo_gaz_menshe_100_kPa_DI);

            runPhase(autoNuOff);
            runPhase(nu1off);
            runPhase(nu2off);
      END_IF;

       IF nu1off.top AND  nu2off.top THEN
  	runPhase(pnsWaitOff);
      END_IF;

      IF waitKran.top AND (NOT kran5Open.top) THEN
  	runUnsuccessful.error:=TRUE;
      END_IF;

      IF pnsWaitOff.top THEN
  	runPhase(autoAvomOff);
  	runPhase(avom1cmdOff);
  	runPhase(avom2cmdOff);
      END_IF;

      IF avom1cmdOff.top AND avom2cmdOff.top THEN
  	 StrAlg.opcCommandsDisabled:=FALSE;
      END_IF;

      StrAlg.isEnded:= avom1cmdOff.top AND avom2cmdOff.top;
  END_IF;

  StrAlg.CanRun := StrAlg.inCanRun;
  StrAlg.OpcCommandsDisabled := StrAlg.inOpcCommandsDisabled;

  (* ---- Если управление с ВУ заблокировано, то  передаем команду из алгоритма ---- *)
  IF StrAlg.inOpcCommandsDisabled THEN
  	StrAlg.inCommand := StrAlg.inCommand_Alg;
  ELSE (* иначе передаем команду с АРМа*)
  	StrAlg.inCommand := StrAlg.inCommand_ARM;
  END_IF;

  _sunpackerCommand(command := StrAlg.inCommand);
  	source := _sunpackerCommand.source;
  	cmd := _sunpackerCommand.cmd;

  IF cmd <> 0 AND lastCmd <> cmd AND (((NOT StrAlg.opcCommandsDisabled) AND source > 0) OR source = 0) then
  	CASE BYTE_TO_INT(cmd) OF
  		(*cmdRun*) 1: 	IF (StrAlg.CanRun) THEN
  					StrAlg.isRuning := TRUE;
  					StrAlg.isEnded := FALSE;
  					StrAlg.hasError := FALSE;
  					(*****************       OnRun       *****************)

                                                    StrAlg.opcCommandsDisabled:=TRUE;
                                                    runIfNotRunningSO(IM.SingleOutputs.Indickaciya_AC_fonar);
                                                    runIfNotRunningSO(IM.SingleOutputs.Rabota_EGPA);
                                                    stopPusk(algoritms);
                                                    algManager.nMode:=ModeGpa.MODE_AO;

                                                    runPhase(waitKran);
                                                    runPhase(runUnsuccessful);

                                                    resetDiProtection(protections.MB);
                                                    resetAiProtection(protections.Vibroskorost_OP_ED_t1_HA);
                                                    resetAiProtection(protections.Vibroskorost_OYP_ED_so_storony_redyctora_t2_HA);
                                                    resetAiProtection(protections.Vibroskorost_OYP_kolesa_ED_t3_HA);
                                                    resetAiProtection(protections.Vibroskorost_OP_kolesa_nagnetatelya_t4_HA);
                                                    resetDiProtection(protections.Kran1sdvig);
                                                    resetDiProtection(protections.Kran2sdvig);

  					cmd_for_Status := cmd;
  					source_for_Status := source;
  					command_error_for_Status := 0;
  				ELSE
  					StrAlg.isRuning := FALSE;
  					StrAlg.isEnded := FALSE;
  					StrAlg.hasError 	:= FALSE;

  					cmd_for_Status := 0;
  					source_for_Status := source;
  					command_error_for_Status := cmd;
  				END_IF;
  		(*cmdReset*) 2: 	StrAlg.isRuning := FALSE;
  				StrAlg.isEnded := FALSE;
  				StrAlg.hasError 	:= FALSE;

                                           (*****************       OnReset       *****************)
                                          protectManager.inCommand:=PMcommand.RestartAllSignaling;
                                          waitReset(IN:=FALSE);
                                          resetIfRunningSO(IM.SingleOutputs.Indickaciya_AC_fonar);
                                          resetIfRunningSO(IM.SingleOutputs.Rabota_EGPA);
                                          resetIfRunning(algoritms.vibegPNS);
                                          algManager.nMode:=ModeGpa.MODE_STOP;
                                          (*impulseSO(Im.singleSignals.Srabotka_BREO);*)

                                          resetPhase(kran4Close);
                                          resetPhase(mvOff);
                                          resetPhase(pnsOn);
                                          resetPhase(kran3bOpen);
                                          resetPhase(kran1Close);
                                          resetPhase(kran2Close);
                                          resetPhase(kran5Open);
                                          resetPhase(autoNuOff);
                                          resetPhase(autoPnsOff);
                                          resetPhase(pInNagLess100);
  	                              resetPhase(autoAvomOff);
                                          resetPhase(avom1cmdOff);
                                          resetPhase(avom2cmdOff);
                                          resetPhase(nu1off);
                                          resetPhase(nu2off);
                                          resetPhase(waitKran);
                                          resetPhase(pnsWaitOff);
                                          resetPhase(runUnsuccessful);

  				cmd_for_Status := cmd;
  				source_for_Status := source;
  				command_error_for_Status := 0;
  	END_CASE;
  	resetCmdTimer(IN := false);
  	resetCmdTimerPriznak := TRUE;
  END_IF;
  lastCmd := cmd;

  resetCmdTimer(IN := resetCmdTimerPriznak, PT := T#5S);
  IF resetCmdTimer.Q THEN
  	resetCmdTimerPriznak := FALSE;
  	source_for_Status := 0;
  	cmd_for_Status := 0;
  	command_error_for_Status := 0;
  END_IF;

  StrAlg.Start:= kran4Close.startStatus
              OR mvOff.startStatus
              OR pnsOn.startStatus
              OR kran3bOpen.startStatus
              OR kran1Close.startStatus
              OR kran2Close.startStatus
              OR kran5Open.startStatus
              OR autoNuOff.startStatus
              OR autoPnsOff.startStatus
              OR pInNagLess100.startStatus
              OR autoAvomOff.startStatus
              OR avom1cmdOff.startStatus
              OR avom2cmdOff.startStatus
              OR nu1off.startStatus
              OR nu2off.startStatus
              OR waitKran.startStatus
              OR pnsWaitOff.startStatus
              OR runUnsuccessful.startStatus;

  StrAlg.Error:= kran4Close.errorStatus
              OR mvOff.errorStatus
              OR pnsOn.errorStatus
              OR kran3bOpen.errorStatus
              OR kran1Close.errorStatus
              OR kran2Close.errorStatus
              OR kran5Open.errorStatus
              OR autoNuOff.errorStatus
              OR autoPnsOff.errorStatus
              OR pInNagLess100.errorStatus
              OR autoAvomOff.errorStatus
              OR avom1cmdOff.errorStatus
              OR avom2cmdOff.errorStatus
              OR nu1off.errorStatus
              OR nu2off.errorStatus
              OR waitKran.errorStatus
              OR pnsWaitOff.errorStatus
              OR runUnsuccessful.errorStatus;

  StrAlg.Top:=   kran4Close.topStatus
              OR mvOff.topStatus
              OR pnsOn.topStatus
              OR kran3bOpen.topStatus
              OR kran1Close.topStatus
              OR kran2Close.topStatus
              OR kran5Open.topStatus
              OR autoNuOff.topStatus
              OR autoPnsOff.topStatus
              OR pInNagLess100.topStatus
              OR autoAvomOff.topStatus
              OR avom1cmdOff.topStatus
              OR avom2cmdOff.topStatus
              OR nu1off.topStatus
              OR nu2off.topStatus
              OR waitKran.topStatus
              OR pnsWaitOff.topStatus
              OR runUnsuccessful.topStatus;

  (*TODO: TYPE PROGRAM CODE HERE*)
  StrAlg.status :=  SHL(BYTE_TO_DWORD(source_for_Status), 29)
  			OR SHL(BYTE_TO_DWORD(cmd_for_Status), 26)
  			OR SHL(BYTE_TO_DWORD(command_error_for_Status), 23)
  			OR SHL(BOOL_TO_DWORD(StrAlg.OpcCommandsDisabled ), 21)
  			OR SHL(BOOL_TO_DWORD(StrAlg.hasError),4)
  			OR SHL(BOOL_TO_DWORD(StrAlg.CanRun),2)
  			OR SHL(BOOL_TO_DWORD(StrAlg.isEnded),1)
  			OR BOOL_TO_DWORD(StrAlg.isRuning);
END_FUNCTION_BLOCK

FUNCTION_BLOCK fb_AlgoritmsManager
  VAR_IN_OUT
    str_AM : struct_AlgoritmsManager;
  END_VAR
  VAR
    onInit : BOOL;
    puskV : BOOL;
  END_VAR
  VAR_EXTERNAL
    ai : AiConfig;
  END_VAR
  VAR
    EoTrig : R_TRIG;
    EoFTrig : F_TRIG;
    PsLampTrig : R_TRIG;
    PsLampFTrig : F_TRIG;
    Ring : R_TRIG;
    Line : R_TRIG;
    statusDualInput : TYPE_statusDualInput;
  END_VAR
  VAR_EXTERNAL
    IM : ImConfig;
    protections : ProtectionsConfig;
    algoritms : AlgoritmsConfig;
    ModeGpa : TYPE_ModeGpa;
  END_VAR

  IF NOT onInit THEN
            DisableAiLimits(ai);
            str_AM.nMode:=ModeGpa.MODE_STOP;
            BlockAllIM(IM);
            runIfNotRunning(algoritms.AutoTen);
  onInit:=TRUE;
  END_IF;

  str_AM.DiscretPS:=anyDiscretPS(IM);
  str_AM.AnalogsPs:=anyAnalogsPs(ai);
  str_AM.ProtectionSignaling:=anyProtectionSignaling(protections);

  EoTrig(CLK := IM.SingleSignals.Srabotka_BREO.Q);
  IF EoTrig.Q THEN
  	stopPusk(algoritms);
  	resetAndDisable(algoritms.Remont);
  	resetAndDisable(algoritms.no);
  	resetAndDisable(algoritms.ao);
  	str_AM.nMode:=ModeGpa.MODE_EO;
  END_IF;
  EoFTrig(CLK := IM.SingleSignals.Srabotka_BREO.Q);
  IF EoFTrig.Q THEN
  	str_AM.nMode:=ModeGpa.MODE_STOP;
  	runIfNotRunning(algoritms.ao);
  END_IF;

  IF (str_AM.ProtectionSignaling OR Im.SingleSignals.AO_KC_ot_SHKC_04M.Q OR Im.SingleSignals.AO_GPA_na_SHY.Q OR Im.SingleSignals.AO_EGPA_ot_PRY.Q )
  	AND NOT((str_AM.mode=ModeGpa.MODE_AO) OR (str_AM.mode=ModeGpa.MODE_EO) OR IM.SingleOutputs.Indickaciya_AC_fonar.Q
            OR (str_AM.mode=ModeGpa.MODE_TESTAZ) OR (str_AM.mode=ModeGpa.MODE_TESTDPMG) OR (str_AM.mode=ModeGpa.MODE_REMONT) OR
            (str_AM.mode=ModeGpa.MODE_TESTPMS))THEN
  		runIfNotRunning(algoritms.ao);
  	str_AM.nMode:=ModeGpa.MODE_AO;
  END_IF;

  IF Im.SingleSignals.NO_GPA_na_SHY.Q  AND algoritms.no.CanRun THEN
  	runIfNotRunning(algoritms.no);
            str_AM.nMode:=ModeGpa.MODE_NO;
  END_IF;

  PsLampTrig(CLK := str_AM.DiscretPS OR str_AM.AnalogsPs);
  IF PsLampTrig.Q THEN
            runIfNotRunningSO(IM.SingleOutputs.Indickaciya_PC_fonar);
  END_IF;
  PsLampFTrig(CLK := str_AM.DiscretPS OR str_AM.AnalogsPs);
  IF PsLampFTrig.Q THEN
            resetIfRunningSO(IM.SingleOutputs.Indickaciya_PC_fonar);
  END_IF;

  IF str_AM.mode = ModeGpa.MODE_WORK_Line OR str_AM.mode = ModeGpa.MODE_WORK_Ring  THEN

  	Ring(CLK:=Im.kran6.onStatus=statusDualInput.STATUS_On);
  	Line(CLK:=Im.kran6.onStatus=statusDualInput.STATUS_Off);

  	IF Ring.Q AND str_AM.mode = ModeGpa.MODE_WORK_Line THEN
  		str_AM.nMode:=ModeGpa.MODE_WORK_Ring;
  	END_IF;
  	IF Line.Q AND str_AM.mode = ModeGpa.MODE_WORK_Ring THEN
  		str_AM.nMode:=ModeGpa.MODE_WORK_Line;
  	END_IF;

  END_IF;

  IF str_AM.mode = ModeGpa.MODE_WORK_Line THEN
            runIfNotRunning(alg:=algoritms.AntiPompag);
  	ELSE
            resetAndDisable(alg:=algoritms.AntiPompag);
  END_IF;

  IF str_AM.nMode<>str_AM.mode THEN
  	str_AM.mode:=str_AM.nMode;
  	CASE str_AM.mode OF
  	(*ModeGpa.MODE_REMONT*)1:
  		stopPusk(algoritms);
  		resetAndDisable(alg:=algoritms.no);
  		resetAndDisable(alg:=algoritms.ao);
  		resetAndDisable(alg:=algoritms.TestProtection);
                      resetAndDisable(alg:=algoritms.testIm);

  	(*ModeGpa.MODE_TESTAZ*)16:
  		stopPusk(algoritms);
  		resetAndDisable(alg:=algoritms.ao);
  		resetAndDisable(alg:=algoritms.no);
                      resetAndDisable(alg:=algoritms.Remont);
                      resetAndDisable(alg:=algoritms.testIm);

            (*ModeGpa.MODE_TESTIM*)15:
                      stopPusk(algoritms);
                      resetAndDisable(alg:=algoritms.Remont);
                      resetAndDisable(alg:=algoritms.TestProtection);

  	(*ModeGpa.MODE_EO*)14:
  		stopPusk(algoritms);
  		resetAndDisable(alg:=algoritms.no);
  		resetAndDisable(alg:=algoritms.ao);
  		resetAndDisable(alg:=algoritms.Remont);
                      resetAndDisable(alg:=algoritms.testIm);
  	(*ModeGpa.MODE_AO*)13:
  		(*//stopPusk();*)
  		resetAndDisable(alg:=algoritms.no);
  		resetAndDisable(alg:=algoritms.Remont);
                      resetAndDisable(alg:=algoritms.testIm);
                      algoritms.VibegPNS.inCanRun:=TRUE;
  	(*ModeGpa.MODE_NO*)12:
  		stopPusk(algoritms);
                      resetAndDisable(alg:=algoritms.testIm);
                      resetAndDisable(alg:=algoritms.Remont);
                      algoritms.VibegPNS.inCanRun:=TRUE;
  		algoritms.ao.inCanRun:=TRUE;
  	(*ModeGpa.MODE_APUSK*)8:
  		resetAndDisable(alg:=algoritms.SemiAutoPusk);
  		resetAndDisable(alg:=algoritms.puskV);
  		resetAndDisable(alg:=algoritms.puskK);
  		resetAndDisable(alg:=algoritms.testdPmg);
  		resetAndDisable(alg:=algoritms.testPms);
  		resetAndDisable(alg:=algoritms.testIm	 );
  		resetAndDisable(alg:=algoritms.ppu);
  		algoritms.no.inCanRun:=TRUE;
  		algoritms.ao.inCanRun:=TRUE;

  	(*ModeGpa.MODE_MPUSK*)9:
  		resetAndDisable(alg:=algoritms.Apusk);
  		resetAndDisable(alg:=algoritms.puskV);
  		resetAndDisable(alg:=algoritms.puskK);
  		resetAndDisable(alg:=algoritms.testdPmg);
  		resetAndDisable(alg:=algoritms.testPms);
  		resetAndDisable(alg:=algoritms.testIm	 );
  		resetAndDisable(alg:=algoritms.ppu);
  		algoritms.no.inCanRun:=TRUE;
                      algoritms.no.inOpcCommandsDisabled:=FALSE;
  		algoritms.ao.inCanRun:=TRUE;
                      algoritms.ao.inOpcCommandsDisabled:=FALSE;

  	(*ModeGpa.MODE_PUSKK*)5:
  		resetAndDisable(alg:=algoritms.Apusk);
  		resetAndDisable(alg:=algoritms.SemiAutoPusk);
  		resetAndDisable(alg:=algoritms.puskV);
  		resetAndDisable(alg:=algoritms.testdPmg);
  		resetAndDisable(alg:=algoritms.testPms);
  		resetAndDisable(alg:=algoritms.ppu);
  		resetAndDisable(alg:=algoritms.testIm	 );
  		algoritms.no.inCanRun:=TRUE;
                      algoritms.no.inOpcCommandsDisabled:=FALSE;
  		algoritms.ao.inCanRun:=TRUE;
                      algoritms.ao.inOpcCommandsDisabled:=FALSE;
  	(*ModeGpa.MODE_PUSKV*)4:
  		resetAndDisable(alg:=algoritms.Apusk);
  		resetAndDisable(alg:=algoritms.SemiAutoPusk);
  		resetAndDisable(alg:=algoritms.puskK);
  		resetAndDisable(alg:=algoritms.testdPmg);
  		resetAndDisable(alg:=algoritms.testPms);
  		resetAndDisable(alg:=algoritms.ppu);
  		resetAndDisable(alg:=algoritms.testIm	 );
  		algoritms.no.inCanRun:=TRUE;
                      algoritms.no.puskV:=TRUE;
                      algoritms.no.inOpcCommandsDisabled:=FALSE;
  		algoritms.ao.inCanRun:=TRUE;
                      algoritms.ao.inOpcCommandsDisabled:=FALSE;

  	(*ModeGpa.MODE_TESTDPMG*)6:
  		resetAndDisable(alg:=algoritms.Apusk);
  		resetAndDisable(alg:=algoritms.SemiAutoPusk);
  		resetAndDisable(alg:=algoritms.puskV);
  		resetAndDisable(alg:=algoritms.puskK);
  		resetAndDisable(alg:=algoritms.testPms);
  		resetAndDisable(alg:=algoritms.ppu);
  		resetAndDisable(alg:=algoritms.testIm	 );
  		algoritms.no.inCanRun:=TRUE;
                      algoritms.no.inOpcCommandsDisabled:=FALSE;
  		algoritms.ao.inCanRun:=TRUE;
                      algoritms.ao.inOpcCommandsDisabled:=FALSE;

  	(*ModeGpa.MODE_TESTPMS*)7:
  		resetAndDisable(alg:=algoritms.Apusk);
  		resetAndDisable(alg:=algoritms.SemiAutoPusk);
  		resetAndDisable(alg:=algoritms.puskV);
  		resetAndDisable(alg:=algoritms.puskK);
  		resetAndDisable(alg:=algoritms.testdPmg);
  		resetAndDisable(alg:=algoritms.ppu);
  		resetAndDisable(alg:=algoritms.testIm	 );
  		algoritms.no.inCanRun:=TRUE;
                      algoritms.no.inOpcCommandsDisabled:=FALSE;
  		algoritms.ao.inCanRun:=TRUE;
                      algoritms.ao.inOpcCommandsDisabled:=FALSE;

  	(*ModeGpa.MODE_WORK_Ring*)10:
  		resetAndDisable(alg:=algoritms.Apusk);
  		resetAndDisable(alg:=algoritms.SemiAutoPusk);
  		resetAndDisable(alg:=algoritms.puskV);
  		resetAndDisable(alg:=algoritms.puskK);
  		resetAndDisable(alg:=algoritms.testdPmg);
  		resetAndDisable(alg:=algoritms.testPms);
  		resetAndDisable(alg:=algoritms.ppu);
  		resetAndDisable(alg:=algoritms.testIm	 );
  		algoritms.no.inCanRun:=TRUE;
                      algoritms.no.inOpcCommandsDisabled:=FALSE;
  		algoritms.ao.inCanRun:=TRUE;
                      algoritms.ao.inOpcCommandsDisabled:=FALSE;

  	(*ModeGpa.MODE_WORK_Line*)11:
  		resetAndDisable(alg:=algoritms.Apusk);
  		resetAndDisable(alg:=algoritms.SemiAutoPusk);
  		resetAndDisable(alg:=algoritms.puskV);
  		resetAndDisable(alg:=algoritms.puskK);
  		resetAndDisable(alg:=algoritms.testdPmg);
  		resetAndDisable(alg:=algoritms.testPms);
  		resetAndDisable(alg:=algoritms.ppu);
  		resetAndDisable(alg:=algoritms.testIm	 );
  		algoritms.no.inCanRun:=TRUE;
                      algoritms.no.inOpcCommandsDisabled:=FALSE;
  		algoritms.ao.inCanRun:=TRUE;
                      algoritms.ao.inOpcCommandsDisabled:=FALSE;

  	(*ModeGpa.MODE_STOP*)2:
  		algoritms.ppu.inCanRun:=TRUE;
                      runIfNotRunning(alg:=algoritms.ppu);
  		algoritms.no.inCanRun:=TRUE;
                      algoritms.no.inOpcCommandsDisabled:=FALSE;
  		algoritms.ao.inCanRun:=TRUE;
                      algoritms.no.puskV:=FALSE;
                      algoritms.ao.inOpcCommandsDisabled:=FALSE;
                      (*UnBlockAllProtections(protections);*)
  		BlockAllIM(IM);
  		algoritms.Remont.inCanRun:=TRUE;
  		algoritms.Remont.inOpcCommandsDisabled:=FALSE;
  		algoritms.testim.inCanRun:=TRUE;
  		algoritms.testim.inOpcCommandsDisabled:=FALSE;
  		algoritms.TestProtection.inCanRun:=TRUE;
  		algoritms.TestProtection.inOpcCommandsDisabled:=FALSE;
                      algoritms.VibegPNS.inCanRun:=FALSE;
  		resetAndDisable(alg:=algoritms.puskV);
  		resetAndDisable(alg:=algoritms.puskK);
  		resetAndDisable(alg:=algoritms.testdPmg);
  		resetAndDisable(alg:=algoritms.testPms);
  	(*ModeGpa.MODE_READY*)3:
  		resetAndDisable(alg:=algoritms.Remont);
  		algoritms.Remont.inOpcCommandsDisabled:=TRUE;
  		resetAndDisable(alg:=algoritms.testim);
  		algoritms.testim.inOpcCommandsDisabled:=TRUE;
  		resetAndDisable(alg:=algoritms.TestProtection);
  		algoritms.TestProtection.inOpcCommandsDisabled:=TRUE;
  	END_CASE;
  END_IF;
END_FUNCTION_BLOCK

FUNCTION_BLOCK OPC_IM_get
  VAR_EXTERNAL
    IM : ImConfig;
    IM_CMN_pump_inCommand_ARM : UINT;
    IM_Kalorifer_ABO_inCommand_ARM : UINT;
    IM_MB_inCommand_ARM : UINT;
    IM_Ten_MB_inCommand_ARM : UINT;
    IM_Ten_kollect_inCommand_ARM : UINT;
    IM_kran1_inCommand_ARM : UINT;
    IM_kran2_inCommand_ARM : UINT;
    IM_kran3b_inCommand_ARM : UINT;
    IM_kran4_inCommand_ARM : UINT;
    IM_kran5_inCommand_ARM : UINT;
    IM_kran6_inCommand_ARM : UINT;
    IM_nu1_inCommand_ARM : UINT;
    IM_nu2_inCommand_ARM : UINT;
    IM_pns_inCommand_ARM : UINT;
    IM_v1_Avom_inCommand_ARM : UINT;
    IM_v2_Avom_inCommand_ARM : UINT;
    IM_v3_Avom_inCommand_ARM : UINT;
    IM_v4_Avom_inCommand_ARM : UINT;
    IM_kran3_inCommand_ARM : UINT;
  END_VAR

  (* OPC Get - IM. Чтение текущих состояний тэгов _______________________________________________________*)

  Im.kran1.inCommand_ARM	:= UINT_TO_WORD(IM_kran1_inCommand_ARM);
  Im.kran2.inCommand_ARM	:= UINT_TO_WORD(IM_kran2_inCommand_ARM);
  Im.kran3.inCommand_ARM	:= UINT_TO_WORD(IM_kran3_inCommand_ARM);
  Im.kran3b.inCommand_ARM	:= UINT_TO_WORD(IM_kran3b_inCommand_ARM);
  Im.kran4.inCommand_ARM	:= UINT_TO_WORD(IM_kran4_inCommand_ARM);
  Im.kran5.inCommand_ARM	:= UINT_TO_WORD(IM_kran5_inCommand_ARM);
  Im.kran6.inCommand_ARM	:= UINT_TO_WORD(IM_kran6_inCommand_ARM);

  Im.pns.inCommand_ARM	:= UINT_TO_WORD(IM_pns_inCommand_ARM);
  Im.Ten_MB.inCommand_ARM	:= UINT_TO_WORD(IM_Ten_MB_inCommand_ARM);
  Im.Ten_kollect.inCommand_ARM	:= UINT_TO_WORD(IM_Ten_kollect_inCommand_ARM);

  Im.v1_Avom.inCommand_ARM	:= UINT_TO_WORD(IM_v1_Avom_inCommand_ARM);
  Im.v2_Avom.inCommand_ARM	:= UINT_TO_WORD(IM_v2_Avom_inCommand_ARM);
  Im.v3_Avom.inCommand_ARM	:= UINT_TO_WORD(IM_v3_Avom_inCommand_ARM);
  Im.v4_Avom.inCommand_ARM	:= UINT_TO_WORD(IM_v4_Avom_inCommand_ARM);

  Im.nu1.inCommand_ARM	:= UINT_TO_WORD(IM_nu1_inCommand_ARM);
  Im.nu2.inCommand_ARM	:= UINT_TO_WORD(IM_nu2_inCommand_ARM);

  Im.Kalorifer_ABO.inCommand_ARM	:= UINT_TO_WORD(IM_Kalorifer_ABO_inCommand_ARM);

  Im.MB.inCommand_ARM	:= UINT_TO_WORD(IM_MB_inCommand_ARM);

  Im.CMN_pump.inCommand_ARM	:= UINT_TO_WORD(IM_CMN_pump_inCommand_ARM);
END_FUNCTION_BLOCK

FUNCTION_BLOCK OPC_IM_set
  VAR_EXTERNAL
    IM : ImConfig;
    IM_SingleSignals_AO_EGPA_ot_PRY_status : UDINT;
    IM_SingleSignals_AO_GPA_na_SHY_status : UDINT;
    IM_SingleSignals_AO_KC_ot_SHKC_04M_status : UDINT;
    IM_SingleSignals_Asinhron_xod_peregryz_status : UDINT;
    IM_SingleSignals_Avar_otkl_viklychatelya_status : UDINT;
    IM_SingleSignals_BEAO_vkl_status : UDINT;
    IM_SingleSignals_Dver_shkafa_otkrita_status : UDINT;
    IM_SingleSignals_EAO_EGPA_ot_PRY_status : UDINT;
    IM_SingleSignals_EAO_GPA_na_SHY_status : UDINT;
    IM_SingleSignals_Gotovnosst_vozb_status : UDINT;
    IM_SingleSignals_NKY_vvod_1_status : UDINT;
    IM_SingleSignals_NKY_vvod_2_status : UDINT;
    IM_SingleSignals_NO_GPA_na_SHY_status : UDINT;
    IM_SingleSignals_Nalichie_220_perem_vhod_v_SHY_status : UDINT;
    IM_SingleSignals_Nalichie_220_post_na_shinah_ypr_ZRY_status : UDINT;
    IM_SingleSignals_Nalichie_220_post_vhod_v_SHY_status : UDINT;
    IM_SingleSignals_Neisprav_BP_10_status : UDINT;
    IM_SingleSignals_Neisprav_BP_1_status : UDINT;
    IM_SingleSignals_Neisprav_BP_2_status : UDINT;
    IM_SingleSignals_Neisprav_BP_3_status : UDINT;
    IM_SingleSignals_Neisprav_BP_4_status : UDINT;
    IM_SingleSignals_Neisprav_BP_5_status : UDINT;
    IM_SingleSignals_Neisprav_BP_6_status : UDINT;
    IM_SingleSignals_Neisprav_BP_7_status : UDINT;
    IM_SingleSignals_Neisprav_BP_8_status : UDINT;
    IM_SingleSignals_Neisprav_BP_9_status : UDINT;
    IM_SingleSignals_Neisprav_cepei_ypr_AVR_pit_vozb_status : UDINT;
    IM_SingleSignals_Net_10_kVt_UcmA_UcmB_status : UDINT;
    IM_SingleSignals_Net_10_kVt_UcmA_UcmC_status : UDINT;
    IM_SingleSignals_Otkl_osn_regylyatora_neisprav_status : UDINT;
    IM_SingleSignals_Potok_masla_posle_ABO_bolshe_status : UDINT;
    IM_SingleSignals_Razreshenie_zagryzki_status : UDINT;
    IM_SingleSignals_SHAVR_1_v_rab_status : UDINT;
    IM_SingleSignals_SHAVR_2_v_rab_status : UDINT;
    IM_SingleSignals_Sbros_srabotki_BREO_status : UDINT;
    IM_SingleSignals_Srabotka_BREO_status : UDINT;
    IM_SingleSignals_dP_gaza_kr_1_status : UDINT;
    IM_SingleSignals_dP_maslo_gaz_menshe_100_kPa_status : UDINT;
    IM_SingleSignals_ostanov_po_zashitam_vozb_avar_status : UDINT;
    IM_SingleSignals_otklon_masla_v_akkym_yplot_status : UDINT;
    IM_CMN_pump_status : UDINT;
    IM_Kalorifer_ABO_status : UDINT;
    IM_MB_status : UDINT;
    IM_Ten_MB_status : UDINT;
    IM_Ten_kollect_status : UDINT;
    IM_kran1_status : UDINT;
    IM_kran2_status : UDINT;
    IM_kran3b_status : UDINT;
    IM_kran4_status : UDINT;
    IM_kran5_status : UDINT;
    IM_kran6_status : UDINT;
    IM_nu1_status : UDINT;
    IM_nu2_status : UDINT;
    IM_pns_status : UDINT;
    IM_v1_Avom_status : UDINT;
    IM_v2_Avom_status : UDINT;
    IM_v3_Avom_status : UDINT;
    IM_v4_Avom_status : UDINT;
    IM_kran3_status : UDINT;
  END_VAR

  (* OPC Set - IM. Запись текущих состояний тэгов _______________________________________________________*)

  IM_kran1_status	:= DWORD_TO_UDINT(Im.kran1.status);
  IM_kran2_status	:= DWORD_TO_UDINT(Im.kran2.status);
  IM_kran3_status	:= DWORD_TO_UDINT(Im.kran3.status);
  IM_kran3b_status	:= DWORD_TO_UDINT(Im.kran3b.status);
  IM_kran4_status	:= DWORD_TO_UDINT(Im.kran4.status);
  IM_kran5_status	:= DWORD_TO_UDINT(Im.kran5.status);
  IM_kran6_status	:= DWORD_TO_UDINT(Im.kran6.status);

  IM_pns_status	:= DWORD_TO_UDINT(Im.pns.status);
  IM_Ten_MB_status	:= DWORD_TO_UDINT(Im.Ten_MB.status);
  IM_Ten_kollect_status	:= DWORD_TO_UDINT(Im.Ten_kollect.status);
  IM_v1_Avom_status	:= DWORD_TO_UDINT(Im.v1_Avom.status);
  IM_v2_Avom_status	:= DWORD_TO_UDINT(Im.v2_Avom.status);
  IM_v3_Avom_status	:= DWORD_TO_UDINT(Im.v3_Avom.status);
  IM_v4_Avom_status	:= DWORD_TO_UDINT(Im.v4_Avom.status);

  IM_nu1_status	:= DWORD_TO_UDINT(Im.nu1.status);
  IM_nu2_status	:= DWORD_TO_UDINT(Im.nu2.status);

  IM_CMN_pump_status         := DWORD_TO_UDINT(Im.CMN_pump.status);
  IM_Kalorifer_ABO_status    := DWORD_TO_UDINT(Im.Kalorifer_ABO.status);
  IM_MB_status               := DWORD_TO_UDINT(Im.MB.status);

  IM_SingleSignals_AO_EGPA_ot_PRY_status            := DWORD_TO_UDINT(Im.SingleSignals.AO_EGPA_ot_PRY.status );
  IM_SingleSignals_AO_GPA_na_SHY_status             := DWORD_TO_UDINT(Im.SingleSignals.AO_GPA_na_SHY.status);
  IM_SingleSignals_AO_KC_ot_SHKC_04M_status         := DWORD_TO_UDINT(Im.SingleSignals.AO_KC_ot_SHKC_04M.status);
  IM_SingleSignals_Asinhron_xod_peregryz_status     := DWORD_TO_UDINT(Im.SingleSignals.Asinhron_xod_peregryz.status);
  IM_SingleSignals_Avar_otkl_viklychatelya_status   := DWORD_TO_UDINT(Im.SingleSignals.Avar_otkl_viklychatelya.status);
  IM_SingleSignals_BEAO_vkl_status                  := DWORD_TO_UDINT(Im.SingleSignals.BEAO_vkl.status );
  IM_SingleSignals_Dver_shkafa_otkrita_status       := DWORD_TO_UDINT(Im.SingleSignals.Dver_shkafa_otkrita.status );
  IM_SingleSignals_EAO_EGPA_ot_PRY_status           := DWORD_TO_UDINT(Im.SingleSignals.EAO_EGPA_ot_PRY.status );
  IM_SingleSignals_EAO_GPA_na_SHY_status            := DWORD_TO_UDINT(Im.SingleSignals.EAO_GPA_na_SHY.status );
  IM_SingleSignals_Gotovnosst_vozb_status           := DWORD_TO_UDINT(Im.SingleSignals.Gotovnosst_vozb.status );

  IM_SingleSignals_NKY_vvod_1_status                            := DWORD_TO_UDINT(Im.SingleSignals.NKY_vvod_1.status );
  IM_SingleSignals_NKY_vvod_2_status                            := DWORD_TO_UDINT(Im.SingleSignals.NKY_vvod_2.status );
  IM_SingleSignals_NO_GPA_na_SHY_status                         := DWORD_TO_UDINT(Im.SingleSignals.NO_GPA_na_SHY.status );
  IM_SingleSignals_Nalichie_220_perem_vhod_v_SHY_status         := DWORD_TO_UDINT(Im.SingleSignals.Nalichie_220_perem_vhod_v_SHY.status );
  IM_SingleSignals_Nalichie_220_post_na_shinah_ypr_ZRY_status   := DWORD_TO_UDINT(Im.SingleSignals.Nalichie_220_post_na_shinah_ypr_ZRY.status );
  IM_SingleSignals_Nalichie_220_post_vhod_v_SHY_status          := DWORD_TO_UDINT(Im.SingleSignals.Nalichie_220_post_vhod_v_SHY.status );
  IM_SingleSignals_Neisprav_cepei_ypr_AVR_pit_vozb_status       := DWORD_TO_UDINT(Im.SingleSignals.Neisprav_cepei_ypr_AVR_pit_vozb.status );
  IM_SingleSignals_Net_10_kVt_UcmA_UcmB_status                  := DWORD_TO_UDINT(Im.SingleSignals.Net_10_kVt_UcmA_UcmB.status );
  IM_SingleSignals_Net_10_kVt_UcmA_UcmC_status                  := DWORD_TO_UDINT(Im.SingleSignals.Net_10_kVt_UcmA_UcmC.status );
  IM_SingleSignals_Otkl_osn_regylyatora_neisprav_status         := DWORD_TO_UDINT(Im.SingleSignals.Otkl_osn_regylyatora_neisprav.status );

  IM_SingleSignals_Neisprav_BP_1_status      := DWORD_TO_UDINT(Im.SingleSignals.Neisprav_BP_1.status );
  IM_SingleSignals_Neisprav_BP_2_status      := DWORD_TO_UDINT(Im.SingleSignals.Neisprav_BP_2.status );
  IM_SingleSignals_Neisprav_BP_3_status      := DWORD_TO_UDINT(Im.SingleSignals.Neisprav_BP_3.status );
  IM_SingleSignals_Neisprav_BP_4_status      := DWORD_TO_UDINT(Im.SingleSignals.Neisprav_BP_4.status );
  IM_SingleSignals_Neisprav_BP_5_status      := DWORD_TO_UDINT(Im.SingleSignals.Neisprav_BP_5.status );
  IM_SingleSignals_Neisprav_BP_6_status      := DWORD_TO_UDINT(Im.SingleSignals.Neisprav_BP_6.status );
  IM_SingleSignals_Neisprav_BP_7_status      := DWORD_TO_UDINT(Im.SingleSignals.Neisprav_BP_7.status );
  IM_SingleSignals_Neisprav_BP_8_status      := DWORD_TO_UDINT(Im.SingleSignals.Neisprav_BP_8.status );
  IM_SingleSignals_Neisprav_BP_9_status      := DWORD_TO_UDINT(Im.SingleSignals.Neisprav_BP_9.status );
  IM_SingleSignals_Neisprav_BP_10_status     := DWORD_TO_UDINT(Im.SingleSignals.Neisprav_BP_10.status );

  IM_SingleSignals_Potok_masla_posle_ABO_bolshe_status      := DWORD_TO_UDINT(Im.SingleSignals.Potok_masla_posle_ABO_bolshe_85_L_min.status );
  IM_SingleSignals_Razreshenie_zagryzki_status              := DWORD_TO_UDINT(Im.SingleSignals.Razreshenie_zagryzki.status );
  IM_SingleSignals_SHAVR_1_v_rab_status                     := DWORD_TO_UDINT(Im.SingleSignals.SHAVR_1_v_rab.status );
  IM_SingleSignals_SHAVR_2_v_rab_status                     := DWORD_TO_UDINT(Im.SingleSignals.SHAVR_2_v_rab.status );
  IM_SingleSignals_Sbros_srabotki_BREO_status               := DWORD_TO_UDINT(Im.SingleSignals.Sbros_srabotki_BREO.status );
  IM_SingleSignals_Srabotka_BREO_status                     := DWORD_TO_UDINT(Im.SingleSignals.Srabotka_BREO.status );
  IM_SingleSignals_dP_gaza_kr_1_status                      := DWORD_TO_UDINT(Im.SingleSignals.dP_gaza_kr_1.status );
  IM_SingleSignals_dP_maslo_gaz_menshe_100_kPa_status       := DWORD_TO_UDINT(Im.SingleSignals.dP_maslo_gaz_menshe_100_kPa.status );
  IM_SingleSignals_ostanov_po_zashitam_vozb_avar_status     := DWORD_TO_UDINT(Im.SingleSignals.ostanov_po_zashitam_vozb_avar.status );
  IM_SingleSignals_otklon_masla_v_akkym_yplot_status        := DWORD_TO_UDINT(Im.SingleSignals.otklon_masla_v_akkym_yplot.status );
END_FUNCTION_BLOCK

FUNCTION_BLOCK OPC_algoritms_get
  VAR_EXTERNAL
    algoritms : AlgoritmsConfig;
    algoritms_AntiPompag_UgolVNA_inCommand_ARM : UINT;
    algoritms_AntiPompag_zapas_inCommand_ARM : UINT;
    algoritms_Apusk_inCommand_ARM : UINT;
    algoritms_AutoAvom_inCommand_ARM : UINT;
    algoritms_AutoPns_inCommand_ARM : UINT;
    algoritms_AutoTen_inCommand_ARM : UINT;
    algoritms_Remont_inCommand_ARM : UINT;
    algoritms_RingToLine_inCommand_ARM : UINT;
    algoritms_SemiAutoPusk_cmdRun1ph_inCommand_ARM : UINT;
    algoritms_SemiAutoPusk_cmdRun2ph_inCommand_ARM : UINT;
    algoritms_SemiAutoPusk_cmdRun3ph_inCommand_ARM : UINT;
    algoritms_SemiAutoPusk_cmdRun4ph_inCommand_ARM : UINT;
    algoritms_SemiAutoPusk_inCommand_ARM : UINT;
    algoritms_TestProtection_inCommand_ARM : UINT;
    algoritms_ao_inCommand_ARM : UINT;
    algoritms_autoNu_Reset_HasNU_inCommand_ARM : UINT;
    algoritms_engineRun_inCommand_ARM : UINT;
    algoritms_filling_inCommand_ARM : UINT;
    algoritms_no_inCommand_ARM : UINT;
    algoritms_ppu_inCommand_ARM : UINT;
    algoritms_puskK_inCommand_ARM : UINT;
    algoritms_puskK_questionFilling_inCommand_ARM : UINT;
    algoritms_puskK_questionUnload_inCommand_ARM : UINT;
    algoritms_puskOilSystem_Ust_dPmg_inCommand_ARM : UINT;
    algoritms_puskOilSystem_inCommand_ARM : UINT;
    algoritms_puskV_inCommand_ARM : UINT;
    algoritms_puskV_questionFilling_inCommand_ARM : UINT;
    algoritms_puskV_questionMVoff_inCommand_ARM : UINT;
    algoritms_testIm_TypeSwitch_inCommand_ARM : UINT;
    algoritms_testIm_inCommand_ARM : UINT;
    algoritms_testPms_algContinue_inCommand_ARM : UINT;
    algoritms_testPms_inCommand_ARM : UINT;
    algoritms_testdPmg_algContinue_inCommand_ARM : UINT;
    algoritms_testdPmg_inCommand_ARM : UINT;
    algoritms_vibegPNS_algContinue_inCommand_ARM : UINT;
    AlgQuestions : AlgoritmsQuestions;
    algoritms_autoNu_inCommand_ARM : UINT;
    algoritms_vibegPNS_inCommand_ARM : UINT;
  END_VAR

  (* OPC Get - algoritms. Чтение текущих состояний тэгов _______________________________________________________*)

  algoritms.ao.inCommand_ARM	:= UINT_TO_WORD(algoritms_ao_inCommand_ARM);

  algoritms.Apusk.inCommand_ARM	:= UINT_TO_WORD(algoritms_Apusk_inCommand_ARM);

  algoritms.AutoAvom.inCommand_ARM	:= UINT_TO_WORD(algoritms_AutoAvom_inCommand_ARM);

  algoritms.autoNu.inCommand_ARM	:= UINT_TO_WORD(algoritms_autoNu_inCommand_ARM);

  algoritms.AutoPns.inCommand_ARM	:= UINT_TO_WORD(algoritms_AutoPns_inCommand_ARM);

  algoritms.engineRun.inCommand_ARM	:= UINT_TO_WORD(algoritms_engineRun_inCommand_ARM);

  algoritms.filling.inCommand_ARM	:= UINT_TO_WORD(algoritms_filling_inCommand_ARM);

  algoritms.no.inCommand_ARM	:= UINT_TO_WORD(algoritms_no_inCommand_ARM);

  algoritms.ppu.inCommand_ARM	:= UINT_TO_WORD(algoritms_ppu_inCommand_ARM);

  AlgQuestions.puskK_questionFilling.inCommand	:= UINT_TO_WORD(algoritms_puskK_questionFilling_inCommand_ARM);
  AlgQuestions.puskK_questionUnload.inCommand	:= UINT_TO_WORD(algoritms_puskK_questionUnload_inCommand_ARM);
  algoritms.puskK.inCommand_ARM	:= UINT_TO_WORD(algoritms_puskK_inCommand_ARM);

  algoritms.puskOilSystem.inCommand_ARM	:= UINT_TO_WORD(algoritms_puskOilSystem_inCommand_ARM);

  AlgQuestions.puskV_questionEngine.inCommand	:= UINT_TO_WORD(algoritms_puskV_questionFilling_inCommand_ARM);
  AlgQuestions.puskV_questionMVoff.inCommand	:= UINT_TO_WORD(algoritms_puskV_questionMVoff_inCommand_ARM);
  algoritms.puskV.inCommand_ARM	:= UINT_TO_WORD(algoritms_puskV_inCommand_ARM);

  algoritms.Remont.inCommand_ARM	:= UINT_TO_WORD(algoritms_Remont_inCommand_ARM);

  algoritms.RingToLine.inCommand_ARM	:= UINT_TO_WORD(algoritms_RingToLine_inCommand_ARM);

  AlgQuestions.SemiAutoPusk_cmdRun1ph.inCommand	:= UINT_TO_WORD(algoritms_SemiAutoPusk_cmdRun1ph_inCommand_ARM);
  AlgQuestions.SemiAutoPusk_cmdRun2ph.inCommand	:= UINT_TO_WORD(algoritms_SemiAutoPusk_cmdRun2ph_inCommand_ARM);
  AlgQuestions.SemiAutoPusk_cmdRun3ph.inCommand	:= UINT_TO_WORD(algoritms_SemiAutoPusk_cmdRun3ph_inCommand_ARM);
  AlgQuestions.SemiAutoPusk_cmdRun4ph.inCommand	:= UINT_TO_WORD(algoritms_SemiAutoPusk_cmdRun4ph_inCommand_ARM);
  algoritms.SemiAutoPusk.inCommand_ARM	:= UINT_TO_WORD(algoritms_SemiAutoPusk_inCommand_ARM);

  AlgQuestions.testdPmg_algContinue.inCommand	:= UINT_TO_WORD(algoritms_testdPmg_algContinue_inCommand_ARM);
  algoritms.testdPmg.inCommand_ARM	:= UINT_TO_WORD(algoritms_testdPmg_inCommand_ARM);

  algoritms.testIm.inCommand_ARM	:= UINT_TO_WORD(algoritms_testIm_inCommand_ARM);

  AlgQuestions.testPms_algContinue.inCommand	:= UINT_TO_WORD(algoritms_testPms_algContinue_inCommand_ARM);
  algoritms.testPms.inCommand_ARM	:= UINT_TO_WORD(algoritms_testPms_inCommand_ARM);

  algoritms.TestProtection.inCommand_ARM	:= UINT_TO_WORD(algoritms_TestProtection_inCommand_ARM);

  AlgQuestions.vibegPNS_algContinue.inCommand	:= UINT_TO_WORD(algoritms_vibegPNS_algContinue_inCommand_ARM);
  algoritms.vibegPNS.inCommand_ARM	:= UINT_TO_WORD(algoritms_vibegPNS_inCommand_ARM);

  algoritms.AutoTen.inCommand_ARM	:= UINT_TO_WORD(algoritms_AutoTen_inCommand_ARM);
END_FUNCTION_BLOCK

FUNCTION_BLOCK OPC_algoritms_set
  VAR_EXTERNAL
    algoritms : AlgoritmsConfig;
    algManager_Mode : UINT;
    algoritms_AutoAvom_status : UDINT;
    algoritms_AutoPns_OffTimer : UINT;
    algoritms_AutoPns_OnTimer : UINT;
    algoritms_AutoPns_status : UDINT;
    algoritms_AutoTen_status : UDINT;
    algoritms_Remont_status : UDINT;
    algoritms_TestProtection_status : UDINT;
    algoritms_autoNu_NotHasRezervNU : BOOL;
    algoritms_autoNu_status : UDINT;
    algoritms_puskOilSystem_Error : UDINT;
    algoritms_puskOilSystem_Start : UDINT;
    algoritms_puskOilSystem_Top : UDINT;
    algoritms_puskOilSystem_status : UDINT;
    algoritms_testIm_status : UDINT;
    algoritms_vibegPNS_Error : UDINT;
    algoritms_vibegPNS_Start : UDINT;
    algoritms_vibegPNS_Top : UDINT;
    algoritms_vibegPNS_algContinue_status : UDINT;
    algoritms_vibegPNS_status : UDINT;
    algoritms_vibegPNS_waitVibeg_timer : UINT;
    protectManager_protectionInRemont : BOOL;
    algManager : struct_AlgoritmsManager;
    protectManager : struct_ProtectionsManager;
    NotHasRezervNU : BOOL;
    AlgTimers : struct_AlgTimers;
    AlgQuestions : AlgoritmsQuestions;
    algoritms_Apusk_Error : UDINT;
    algoritms_Apusk_Start : UDINT;
    algoritms_Apusk_Top : UDINT;
    algoritms_Apusk_status : UDINT;
    algoritms_RingToLine_Error : UDINT;
    algoritms_RingToLine_Start : UDINT;
    algoritms_RingToLine_Top : UDINT;
    algoritms_RingToLine_status : UDINT;
    algoritms_SemiAutoPusk_Error : UDINT;
    algoritms_SemiAutoPusk_Start : UDINT;
    algoritms_SemiAutoPusk_Top : UDINT;
    algoritms_SemiAutoPusk_cmdRun1ph_status : UDINT;
    algoritms_SemiAutoPusk_cmdRun2ph_status : UDINT;
    algoritms_SemiAutoPusk_cmdRun3ph_status : UDINT;
    algoritms_SemiAutoPusk_cmdRun4ph_status : UDINT;
    algoritms_SemiAutoPusk_status : UDINT;
    algoritms_ao_Error : UDINT;
    algoritms_ao_Start : UDINT;
    algoritms_ao_Top : UDINT;
    algoritms_ao_status : UDINT;
    algoritms_ao_waitKran_timer : UINT;
    algoritms_engineRun_BreakPuskTimer_timer : UINT;
    algoritms_engineRun_Error : UDINT;
    algoritms_engineRun_Start : UDINT;
    algoritms_engineRun_Top : UDINT;
    algoritms_engineRun_status : UDINT;
    algoritms_filling_BreakPuskTimer_timer : UINT;
    algoritms_filling_Error : UDINT;
    algoritms_filling_Start : UDINT;
    algoritms_filling_Top : UDINT;
    algoritms_filling_status : UDINT;
    algoritms_filling_waitAfterKran4_timer : UINT;
    algoritms_filling_waitAfterKran5_timer : UINT;
    algoritms_no_Error : UDINT;
    algoritms_no_Start : UDINT;
    algoritms_no_Top : UDINT;
    algoritms_no_status : UDINT;
    algoritms_no_waitCloseKran_timer : UINT;
    algoritms_ppu_Error : UDINT;
    algoritms_ppu_Start : UDINT;
    algoritms_ppu_Top : UDINT;
    algoritms_ppu_status : UDINT;
    algoritms_puskK_Error : UDINT;
    algoritms_puskK_Start : UDINT;
    algoritms_puskK_Top : UDINT;
    algoritms_puskK_questionFilling_status : UDINT;
    algoritms_puskK_questionUnload_status : UDINT;
    algoritms_puskK_status : UDINT;
    algoritms_puskK_wait720_timer : UINT;
    algoritms_puskOilSystem_BreakPuskTimer_Poil_timer : UINT;
    algoritms_puskOilSystem_BreakPuskTimer_dPmg_timer : UINT;
    algoritms_puskV_Error : UDINT;
    algoritms_puskV_Start : UDINT;
    algoritms_puskV_Top : UDINT;
    algoritms_puskV_questionFilling_status : UDINT;
    algoritms_puskV_questionMVoff_status : UDINT;
    algoritms_puskV_status : UDINT;
    algoritms_puskV_wait600_timer : UINT;
    algoritms_testPms_BreakTest_timer : UINT;
    algoritms_testPms_Error : UDINT;
    algoritms_testPms_Start : UDINT;
    algoritms_testPms_Top : UDINT;
    algoritms_testPms_algContinue_status : UDINT;
    algoritms_testPms_status : UDINT;
    algoritms_testdPmg_BreakTest_timer : UINT;
    algoritms_testdPmg_Error : UDINT;
    algoritms_testdPmg_Start : UDINT;
    algoritms_testdPmg_Top : UDINT;
    algoritms_testdPmg_algContinue_status : UDINT;
    algoritms_testdPmg_status : UDINT;
  END_VAR

  (* OPC Set - algoritms. Запись текущих состояний тэгов _______________________________________________________*)

  algManager_Mode := algManager.mode;

  protectManager_protectionInRemont:= protectManager.protectionInRemont;

  algoritms_autoNu_NotHasRezervNU:= NotHasRezervNU;

  algoritms_no_Start	:= DWORD_TO_UDINT(algoritms.no.Start);
  algoritms_no_Error	:= DWORD_TO_UDINT(algoritms.no.Error);
  algoritms_no_Top	:= DWORD_TO_UDINT(algoritms.no.Top);
  algoritms_no_status	:= DWORD_TO_UDINT(algoritms.no.status);
  algoritms_no_waitCloseKran_timer	:= AlgTimers.NO_waitCloseKran;

  algoritms_ao_Start	:= DWORD_TO_UDINT(algoritms.ao.Start);
  algoritms_ao_Error	:= DWORD_TO_UDINT(algoritms.ao.Error);
  algoritms_ao_Top	:= DWORD_TO_UDINT(algoritms.ao.Top);
  algoritms_ao_status	:= DWORD_TO_UDINT(algoritms.ao.status);
  algoritms_ao_waitKran_timer	:= AlgTimers.AO_waitKran;

  algoritms_vibegPNS_Start		:= DWORD_TO_UDINT(algoritms.vibegPNS.Start);
  algoritms_vibegPNS_Error		:= DWORD_TO_UDINT(algoritms.vibegPNS.Error);
  algoritms_vibegPNS_Top		:= DWORD_TO_UDINT(algoritms.vibegPNS.Top);
  algoritms_vibegPNS_status		:= DWORD_TO_UDINT(algoritms.vibegPNS.status);
  algoritms_vibegPNS_waitVibeg_timer	:= AlgTimers.vibegPNS_Timer;
  algoritms_vibegPNS_algContinue_status	:= DWORD_TO_UDINT(AlgQuestions.vibegPNS_algContinue.status);

  algoritms_testPms_Start		:= DWORD_TO_UDINT(algoritms.testPms.Start);
  algoritms_testPms_Error		:= DWORD_TO_UDINT(algoritms.testPms.Error);
  algoritms_testPms_Top		:= DWORD_TO_UDINT(algoritms.testPms.Top);
  algoritms_testPms_status		:= DWORD_TO_UDINT(algoritms.testPms.status);
  algoritms_testPms_algContinue_status	:= DWORD_TO_UDINT(AlgQuestions.testPms_algContinue.status);
  algoritms_testPms_BreakTest_timer	:= AlgTimers.testPms_BreakTest;

  algoritms_testdPmg_Start		:= DWORD_TO_UDINT(algoritms.testdPmg.Start);
  algoritms_testdPmg_Error		:= DWORD_TO_UDINT(algoritms.testdPmg.Error);
  algoritms_testdPmg_Top		:= DWORD_TO_UDINT(algoritms.testdPmg.Top);
  algoritms_testdPmg_status		:= DWORD_TO_UDINT(algoritms.testdPmg.status);
  algoritms_testdPmg_algContinue_status	:= DWORD_TO_UDINT(AlgQuestions.testdPmg_algContinue.status);
  algoritms_testdPmg_BreakTest_timer	:= AlgTimers.testdPmg_BreakTest;

  algoritms_testIm_status	:= DWORD_TO_UDINT(algoritms.testIm.status);

  algoritms_ppu_status	:= DWORD_TO_UDINT(algoritms.ppu.status);
  algoritms_ppu_Start	          := DWORD_TO_UDINT(algoritms.ppu.Start);
  algoritms_ppu_Error	          := DWORD_TO_UDINT(algoritms.ppu.Error);
  algoritms_ppu_Top	          := DWORD_TO_UDINT(algoritms.ppu.Top);

  algoritms_puskOilSystem_status			:= DWORD_TO_UDINT(algoritms.puskOilSystem.status);
  algoritms_puskOilSystem_Start				:= DWORD_TO_UDINT(algoritms.puskOilSystem.Start);
  algoritms_puskOilSystem_Error				:= DWORD_TO_UDINT(algoritms.puskOilSystem.Error);
  algoritms_puskOilSystem_Top				:= DWORD_TO_UDINT(algoritms.puskOilSystem.Top);
  algoritms_puskOilSystem_BreakPuskTimer_Poil_timer	          := AlgTimers.puskOilSystem_BreakPuskTimer_Poil;

  algoritms_engineRun_status			:= DWORD_TO_UDINT(algoritms.engineRun.status);
  algoritms_engineRun_Start			:= DWORD_TO_UDINT(algoritms.engineRun.Start);
  algoritms_engineRun_Error			:= DWORD_TO_UDINT(algoritms.engineRun.Error);
  algoritms_engineRun_Top			:= DWORD_TO_UDINT(algoritms.engineRun.Top);
  algoritms_engineRun_BreakPuskTimer_timer	:= AlgTimers.engineRun_BreakPuskTimer;

  algoritms_filling_status		:= DWORD_TO_UDINT(algoritms.filling.status);
  algoritms_filling_Start		:= DWORD_TO_UDINT(algoritms.filling.Start);
  algoritms_filling_Error		:= DWORD_TO_UDINT(algoritms.filling.Error);
  algoritms_filling_Top		:= DWORD_TO_UDINT(algoritms.filling.Top);
  algoritms_filling_BreakPuskTimer_timer	:= AlgTimers.filling_BreakPuskTimer;
  algoritms_filling_waitAfterKran4_timer	:= AlgTimers.filling_waitAfterKran4;
  algoritms_filling_waitAfterKran5_timer	:= AlgTimers.filling_waitAfterKran5;

  algoritms_RingToLine_status	:= DWORD_TO_UDINT(algoritms.RingToLine.status);
  algoritms_RingToLine_Start	:= DWORD_TO_UDINT(algoritms.RingToLine.Start);
  algoritms_RingToLine_Error	:= DWORD_TO_UDINT(algoritms.RingToLine.Error);
  algoritms_RingToLine_Top	:= DWORD_TO_UDINT(algoritms.RingToLine.Top);

  algoritms_puskK_status	            := DWORD_TO_UDINT(algoritms.puskK.status);
  algoritms_puskK_Start	            := DWORD_TO_UDINT(algoritms.puskK.Start);
  algoritms_puskK_Error	            := DWORD_TO_UDINT(algoritms.puskK.Error);
  algoritms_puskK_Top	                      := DWORD_TO_UDINT(algoritms.puskK.Top);
  algoritms_puskK_wait720_timer	            := AlgTimers.puskK_wait720;
  algoritms_puskK_questionFilling_status	  := DWORD_TO_UDINT(AlgQuestions.puskK_questionFilling.status);
  algoritms_puskK_questionUnload_status	  := DWORD_TO_UDINT(AlgQuestions.puskK_questionUnload.status);

  algoritms_puskV_status	          := DWORD_TO_UDINT(algoritms.puskV.status);
  algoritms_puskV_Start	          := DWORD_TO_UDINT(algoritms.puskV.Start);
  algoritms_puskV_Error	          := DWORD_TO_UDINT(algoritms.puskV.Error);
  algoritms_puskV_Top	                    := DWORD_TO_UDINT(algoritms.puskV.Top);
  algoritms_puskV_wait600_timer	          := AlgTimers.puskV_wait600;
  algoritms_puskV_questionFilling_status	:= DWORD_TO_UDINT(AlgQuestions.puskV_questionEngine.status);
  algoritms_puskV_questionMVoff_status	:= DWORD_TO_UDINT(AlgQuestions.puskV_questionMVoff.status);

  algoritms_Apusk_status	:= DWORD_TO_UDINT(algoritms.Apusk.status);
  algoritms_Apusk_Start	:= DWORD_TO_UDINT(algoritms.Apusk.Start);
  algoritms_Apusk_Error	:= DWORD_TO_UDINT(algoritms.Apusk.Error);
  algoritms_Apusk_Top	          := DWORD_TO_UDINT(algoritms.Apusk.Top);

  algoritms_SemiAutoPusk_status	:= DWORD_TO_UDINT(algoritms.SemiAutoPusk.status);
  algoritms_SemiAutoPusk_Start	:= DWORD_TO_UDINT(algoritms.SemiAutoPusk.Start);
  algoritms_SemiAutoPusk_Error	:= DWORD_TO_UDINT(algoritms.SemiAutoPusk.Error);
  algoritms_SemiAutoPusk_Top	:= DWORD_TO_UDINT(algoritms.SemiAutoPusk.Top);
  algoritms_SemiAutoPusk_cmdRun1ph_status	:= DWORD_TO_UDINT(AlgQuestions.SemiAutoPusk_cmdRun1ph.status);
  algoritms_SemiAutoPusk_cmdRun2ph_status	:= DWORD_TO_UDINT(AlgQuestions.SemiAutoPusk_cmdRun2ph.status);
  algoritms_SemiAutoPusk_cmdRun3ph_status	:= DWORD_TO_UDINT(AlgQuestions.SemiAutoPusk_cmdRun3ph.status);
  algoritms_SemiAutoPusk_cmdRun4ph_status	:= DWORD_TO_UDINT(AlgQuestions.SemiAutoPusk_cmdRun4ph.status);

  algoritms_AutoPns_status	:= DWORD_TO_UDINT(algoritms.AutoPns.status);
  algoritms_AutoPns_OnTimer	:= AlgTimers.AutoPns_OnTimer;
  algoritms_AutoPns_OffTimer	:= AlgTimers.AutoPns_OffTimer;

  algoritms_autoNu_status	:= DWORD_TO_UDINT(algoritms.autoNu.status);

  algoritms_AutoAvom_status	:= DWORD_TO_UDINT(algoritms.AutoAvom.status);

  algoritms_TestProtection_status	:= DWORD_TO_UDINT(algoritms.TestProtection.status);

  algoritms_Remont_status	:= DWORD_TO_UDINT(algoritms.Remont.status);

  algoritms_AutoTen_status	:= DWORD_TO_UDINT(algoritms.AutoTen.status);
END_FUNCTION_BLOCK

FUNCTION_BLOCK RemontAlg
  VAR_IN_OUT
    StrAlg : struct_Alg;
  END_VAR
  VAR
    _sunpackerCommand : fb_sunpackerCommand;
    source : BYTE;
    cmd : BYTE;
    lastCmd : BYTE;
    source_for_Status : BYTE;
    cmd_for_Status : BYTE;
    command_error_for_Status : BYTE;
    resetCmdTimer : TON;
    resetCmdTimerPriznak : BOOL;
  END_VAR
  VAR_EXTERNAL
    protectManager : struct_ProtectionsManager;
    algManager : struct_AlgoritmsManager;
    ModeGpa : TYPE_ModeGpa;
    PMcommand : TYPE_CommandsPotectionsManager;
    IM : ImConfig;
  END_VAR

  StrAlg.CanRun := StrAlg.inCanRun;
  StrAlg.OpcCommandsDisabled := StrAlg.inOpcCommandsDisabled;

  (* ---- Если управление с ВУ заблокировано, то передаем команду из алгоритма ---- *)
  IF StrAlg.inOpcCommandsDisabled THEN
  	StrAlg.inCommand := StrAlg.inCommand_Alg;
  ELSE (* иначе передаем команду с АРМа*)
  	StrAlg.inCommand := StrAlg.inCommand_ARM;
  END_IF;

  _sunpackerCommand(command := StrAlg.inCommand);
  	source := _sunpackerCommand.source;
  	cmd := _sunpackerCommand.cmd;

  IF cmd <> 0 AND lastCmd <> cmd AND (((NOT StrAlg.opcCommandsDisabled) AND source > 0) OR source = 0) then
  	CASE BYTE_TO_INT(cmd) OF
  		(*cmdRun*) 1: 	IF (StrAlg.CanRun) THEN
  					StrAlg.isRuning := TRUE;
  					StrAlg.isEnded := FALSE;
  					StrAlg.hasError 	:= FALSE;
                                               (*****************       OnRun       *****************)
                                                        algManager.nMode:=ModeGpa.MODE_REMONT;
                                                        protectManager.inCommand:=PMcommand.ResetAllProtections;
  					    UnBlockAllIM(IM);
                                                    (*StrAlg.inOpcCommandsDisabled:=FALSE;*)
  					cmd_for_Status := cmd;
  					source_for_Status := source;
  					command_error_for_Status := 0;
  				ELSE
  					StrAlg.isRuning := FALSE;
  					StrAlg.isEnded := FALSE;
  					StrAlg.hasError 	:= FALSE;

  					cmd_for_Status := 0;
  					source_for_Status := source;
  					command_error_for_Status := cmd;
  				END_IF;
  		(*cmdReset*) 2: 	StrAlg.isRuning := FALSE;
  				StrAlg.isEnded := FALSE;
  				StrAlg.hasError 	:= FALSE;
                                          (*****************       OnReset       *****************)
                                                    BlockAllIM(IM);
                                                    protectManager.inCommand:=PMcommand.RestartAllProtections;
                                                    algManager.nMode:=ModeGpa.MODE_STOP;

  				cmd_for_Status := cmd;
  				source_for_Status := source;
  				command_error_for_Status := 0;
  	END_CASE;
  	resetCmdTimer(IN := false);
  	resetCmdTimerPriznak := TRUE;
  END_IF;
  lastCmd := cmd;

  resetCmdTimer(IN := resetCmdTimerPriznak, PT := T#5S);
  IF resetCmdTimer.Q THEN
  	resetCmdTimerPriznak := FALSE;
  	source_for_Status := 0;
  	cmd_for_Status := 0;
  	command_error_for_Status := 0;
  END_IF;

  StrAlg.status :=  SHL(BYTE_TO_DWORD(source_for_Status), 29)
  			OR SHL(BYTE_TO_DWORD(cmd_for_Status), 26)
  			OR SHL(BYTE_TO_DWORD(command_error_for_Status), 23)
  			OR SHL(BOOL_TO_DWORD(StrAlg.OpcCommandsDisabled ), 21)
  			OR SHL(BOOL_TO_DWORD(StrAlg.hasError),4)
  			OR SHL(BOOL_TO_DWORD(StrAlg.CanRun),2)
  			OR SHL(BOOL_TO_DWORD(StrAlg.isEnded),1)
  			OR BOOL_TO_DWORD(StrAlg.isRuning);
END_FUNCTION_BLOCK

FUNCTION_BLOCK TestImAlg
  VAR_IN_OUT
    StrAlg : struct_Alg;
  END_VAR
  VAR
    _sunpackerCommand : fb_sunpackerCommand;
    source : BYTE;
    cmd : BYTE;
    lastCmd : BYTE;
    source_for_Status : BYTE;
    cmd_for_Status : BYTE;
    command_error_for_Status : BYTE;
    resetCmdTimer : TON;
    resetCmdTimerPriznak : BOOL;
  END_VAR
  VAR_EXTERNAL
    protectManager : struct_ProtectionsManager;
    algManager : struct_AlgoritmsManager;
    ModeGpa : TYPE_ModeGpa;
    PMcommand : TYPE_CommandsPotectionsManager;
    IM : ImConfig;
  END_VAR

  StrAlg.CanRun := StrAlg.inCanRun;
  StrAlg.OpcCommandsDisabled := StrAlg.inOpcCommandsDisabled;

  (* ---- Если управление с ВУ заблокировано, то передаем команду из алгоритма ---- *)
  IF StrAlg.inOpcCommandsDisabled THEN
  	StrAlg.inCommand := StrAlg.inCommand_Alg;
  ELSE (* иначе передаем команду с АРМа*)
  	StrAlg.inCommand := StrAlg.inCommand_ARM;
  END_IF;

  _sunpackerCommand(command := StrAlg.inCommand);
  	source := _sunpackerCommand.source;
  	cmd := _sunpackerCommand.cmd;

  IF cmd <> 0 AND lastCmd <> cmd AND (((NOT StrAlg.opcCommandsDisabled) AND source > 0) OR source = 0) then
  	CASE BYTE_TO_INT(cmd) OF
  		(*cmdRun*) 1: 	IF (StrAlg.CanRun) THEN
  					StrAlg.isRuning := TRUE;
  					StrAlg.isEnded := FALSE;
  					StrAlg.hasError 	:= FALSE;
                                               (*****************       OnRun       *****************)

                                                        algManager.nMode:=ModeGpa.MODE_TESTIM;
  					    UnBlockAllIM(IM);

                                                    (*StrAlg.inOpcCommandsDisabled:=FALSE;*)
  					cmd_for_Status := cmd;
  					source_for_Status := source;
  					command_error_for_Status := 0;
  				ELSE
  					StrAlg.isRuning := FALSE;
  					StrAlg.isEnded := FALSE;
  					StrAlg.hasError 	:= FALSE;

  					cmd_for_Status := 0;
  					source_for_Status := source;
  					command_error_for_Status := cmd;
  				END_IF;
  		(*cmdReset*) 2: 	StrAlg.isRuning := FALSE;
  				StrAlg.isEnded := FALSE;
  				StrAlg.hasError 	:= FALSE;
                                          (*****************       OnReset       *****************)
                                                    BlockAllIM(IM);
                                                    algManager.nMode:=ModeGpa.MODE_STOP;

  				cmd_for_Status := cmd;
  				source_for_Status := source;
  				command_error_for_Status := 0;
  	END_CASE;
  	resetCmdTimer(IN := false);
  	resetCmdTimerPriznak := TRUE;
  END_IF;
  lastCmd := cmd;

  resetCmdTimer(IN := resetCmdTimerPriznak, PT := T#5S);
  IF resetCmdTimer.Q THEN
  	resetCmdTimerPriznak := FALSE;
  	source_for_Status := 0;
  	cmd_for_Status := 0;
  	command_error_for_Status := 0;
  END_IF;
